C09156=1172.373,-59.206,-43.049,179.363,5.809,149.223
C09157=1172.378,-59.456,-43.037,179.360,5.808,149.223
C09158=1172.384,-59.705,-43.026,179.358,5.808,149.224
C09159=1172.389,-59.955,-43.015,179.356,5.808,149.225
C09160=1172.394,-60.205,-43.003,179.354,5.807,149.225
C09161=1172.400,-60.454,-42.993,179.351,5.807,149.226
C09162=1172.404,-60.704,-42.982,179.349,5.806,149.227
C09163=1172.410,-60.953,-42.971,179.347,5.807,149.227
C09164=1172.415,-61.203,-42.960,179.344,5.806,149.228
C09165=1172.420,-61.453,-42.948,179.342,5.805,149.228
C09166=1172.426,-61.702,-42.938,179.339,5.805,149.229
C09167=1172.430,-61.952,-42.927,179.337,5.805,149.230
C09168=1172.436,-62.203,-42.916,179.335,5.805,149.230
C09169=1172.441,-62.452,-42.905,179.333,5.804,149.231
C09170=1172.446,-62.702,-42.894,179.331,5.804,149.232
C09171=1172.452,-62.951,-42.883,179.328,5.803,149.232
C09172=1172.456,-63.200,-42.872,179.326,5.803,149.233
C09173=1172.462,-63.451,-42.861,179.323,5.803,149.233
C09174=1172.467,-63.700,-42.850,179.321,5.803,149.234
C09175=1172.472,-63.950,-42.839,179.319,5.802,149.235
C09176=1172.478,-64.199,-42.828,179.317,5.801,149.235
C09177=1172.483,-64.449,-42.818,179.314,5.801,149.236
C09178=1172.488,-64.699,-42.806,179.312,5.801,149.236
C09179=1172.494,-64.949,-42.796,179.310,5.801,149.237
C09180=1172.498,-65.198,-42.784,179.307,5.800,149.238
C09181=1172.504,-65.448,-42.774,179.305,5.800,149.238
C09182=1172.509,-65.698,-42.764,179.303,5.800,149.239
C09183=1172.515,-65.947,-42.752,179.301,5.799,149.239
C09184=1172.520,-66.198,-42.742,179.298,5.799,149.240
C09185=1172.525,-66.447,-42.730,179.296,5.799,149.241
C09186=1172.530,-66.697,-42.720,179.294,5.798,149.241
C09187=1172.535,-66.946,-42.709,179.291,5.798,149.242
C09188=1172.541,-67.196,-42.699,179.289,5.798,149.242
C09189=1172.546,-67.446,-42.688,179.287,5.797,149.243
C09190=1172.552,-67.695,-42.677,179.284,5.796,149.244
C09191=1172.557,-67.946,-42.666,179.282,5.797,149.244
C09192=1172.562,-68.195,-42.655,179.280,5.796,149.245
C09193=1172.567,-68.445,-42.644,179.278,5.796,149.245
C09194=1172.573,-68.694,-42.634,179.275,5.795,149.246
C09195=1172.577,-68.944,-42.623,179.273,5.795,149.247
C09196=1172.583,-69.194,-42.613,179.271,5.795,149.247
C09197=1172.588,-69.444,-42.602,179.268,5.794,149.248
C09198=1172.593,-69.693,-42.591,179.266,5.794,149.249
C09199=1172.598,-69.943,-42.581,179.264,5.794,149.249
C09200=1172.605,-70.193,-42.570,179.261,5.793,149.250
C09201=1172.609,-70.442,-42.559,179.259,5.794,149.250
C09202=1172.615,-70.692,-42.548,179.257,5.793,149.251
C09203=1172.620,-70.942,-42.538,179.255,5.792,149.252
C09204=1172.625,-71.191,-42.527,179.253,5.792,149.252
C09205=1172.630,-71.441,-42.516,179.250,5.792,149.253
C09206=1172.636,-71.691,-42.506,179.248,5.791,149.253
C09207=1172.641,-71.941,-42.495,179.246,5.792,149.254
C09208=1172.646,-72.190,-42.485,179.244,5.791,149.254
C09209=1172.651,-72.440,-42.474,179.241,5.790,149.255
C09210=1172.657,-72.690,-42.464,179.238,5.790,149.256
C09211=1172.661,-72.940,-42.452,179.237,5.790,149.256
C09212=1172.667,-73.189,-42.442,179.234,5.790,149.257
C09213=1172.672,-73.439,-42.432,179.232,5.789,149.258
C09214=1172.677,-73.689,-42.422,179.230,5.789,149.258
C09215=1172.683,-73.938,-42.411,179.228,5.788,149.259
C09216=1172.688,-74.188,-42.400,179.225,5.788,149.259
C09217=1172.693,-74.438,-42.390,179.224,5.788,149.260
C09218=1172.698,-74.688,-42.379,179.221,5.788,149.261
C09219=1172.704,-74.937,-42.369,179.219,5.787,149.261
C09220=1172.709,-75.188,-42.358,179.217,5.787,149.262
C09221=1172.714,-75.437,-42.348,179.214,5.787,149.263
C09222=1172.720,-75.708,-42.336,179.212,5.786,149.263
C09223=1172.726,-75.979,-42.325,179.209,5.786,149.264
C09224=1172.732,-76.250,-42.314,179.207,5.786,149.264
C09225=1172.737,-76.521,-42.302,179.204,5.786,149.265
C09226=1172.742,-76.771,-42.292,179.202,5.785,149.266
C09227=1172.748,-77.020,-42.282,179.200,5.785,149.266
C09228=1172.753,-77.270,-42.271,179.198,5.784,149.267
C09229=1172.759,-77.520,-42.261,179.195,5.784,149.268
C09230=1172.764,-77.770,-42.250,179.194,5.784,149.268
C09231=1172.769,-78.020,-42.240,179.191,5.784,149.269
C09232=1172.775,-78.269,-42.230,179.189,5.783,149.269
C09233=1172.779,-78.519,-42.219,179.187,5.783,149.270
C09234=1172.785,-78.768,-42.209,179.184,5.783,149.270
C09235=1172.790,-79.019,-42.198,179.182,5.782,149.271
C09236=1172.796,-79.268,-42.188,179.180,5.783,149.272
C09237=1172.801,-79.518,-42.178,179.177,5.782,149.272
C09238=1172.805,-79.768,-42.168,179.175,5.781,149.273
C09239=1172.811,-80.017,-42.157,179.173,5.781,149.274
C09240=1172.817,-80.267,-42.147,179.171,5.781,149.274
C09241=1172.822,-80.517,-42.137,179.168,5.780,149.275
C09242=1172.827,-80.767,-42.126,179.166,5.781,149.275
C09243=1172.833,-81.016,-42.116,179.164,5.780,149.276
C09244=1172.838,-81.266,-42.106,179.161,5.779,149.277
C09245=1172.843,-81.516,-42.096,179.160,5.779,149.277
C09246=1172.848,-81.766,-42.085,179.157,5.779,149.278
C09247=1172.853,-82.015,-42.075,179.155,5.778,149.278
C09248=1172.859,-82.265,-42.065,179.153,5.779,149.279
C09249=1172.864,-82.515,-42.054,179.151,5.778,149.279
C09250=1172.870,-82.765,-42.044,179.149,5.778,149.280
C09251=1172.874,-83.014,-42.035,179.146,5.777,149.281
C09252=1172.879,-83.264,-42.024,179.144,5.777,149.281
C09253=1172.885,-83.514,-42.014,179.142,5.777,149.282
C09254=1172.891,-83.763,-42.004,179.139,5.777,149.283
C09255=1172.896,-84.013,-41.993,179.137,5.776,149.283
C09256=1172.900,-84.263,-41.983,179.135,5.776,149.284
C09257=1172.906,-84.512,-41.973,179.133,5.776,149.284
C09258=1172.912,-84.762,-41.963,179.130,5.775,149.285
C09259=1172.917,-85.012,-41.952,179.128,5.775,149.286
C09260=1172.922,-85.262,-41.943,179.126,5.775,149.286
C09261=1172.927,-85.511,-41.933,179.124,5.775,149.287
C09262=1172.932,-85.762,-41.923,179.122,5.774,149.287
C09263=1172.938,-86.011,-41.913,179.119,5.774,149.288
C09264=1172.944,-86.261,-41.902,179.118,5.774,149.289
C09265=1172.948,-86.510,-41.893,179.115,5.774,149.289
C09266=1172.953,-86.760,-41.882,179.113,5.773,149.290
C09267=1172.959,-87.010,-41.872,179.111,5.773,149.290
C09268=1172.964,-87.260,-41.863,179.108,5.772,149.291
C09269=1172.969,-87.510,-41.852,179.106,5.773,149.292
C09270=1172.975,-87.759,-41.842,179.104,5.772,149.292
C09271=1172.980,-88.009,-41.832,179.101,5.772,149.293
C09272=1172.985,-88.258,-41.822,179.100,5.772,149.293
C09273=1172.990,-88.508,-41.812,179.097,5.771,149.294
C09274=1172.996,-88.759,-41.802,179.096,5.771,149.294
C09275=1173.001,-89.008,-41.793,179.093,5.771,149.295
C09276=1173.007,-89.257,-41.783,179.091,5.770,149.296
C09277=1173.012,-89.508,-41.772,179.089,5.770,149.296
C09278=1173.016,-89.757,-41.762,179.086,5.770,149.297
C09279=1173.022,-90.007,-41.753,179.084,5.769,149.298
C09280=1173.028,-90.257,-41.743,179.082,5.769,149.298
C09281=1173.032,-90.507,-41.733,179.080,5.769,149.299
C09282=1173.038,-90.756,-41.722,179.078,5.769,149.299
C09283=1173.044,-91.006,-41.713,179.075,5.769,149.300
C09284=1173.049,-91.255,-41.703,179.073,5.768,149.300
C09285=1173.054,-91.505,-41.693,179.071,5.768,149.301
C09286=1173.059,-91.755,-41.683,179.069,5.767,149.302
C09287=1173.064,-92.005,-41.674,179.067,5.768,149.302
C09288=1173.070,-92.255,-41.663,179.065,5.767,149.303
C09289=1173.076,-92.504,-41.653,179.062,5.767,149.304
C09290=1173.081,-92.754,-41.644,179.060,5.767,149.304
C09291=1173.086,-93.004,-41.634,179.058,5.766,149.305
C09292=1173.091,-93.253,-41.624,179.056,5.766,149.305
C09293=1173.097,-93.504,-41.615,179.053,5.766,149.306
C09294=1173.102,-93.753,-41.604,179.051,5.765,149.306
C09295=1173.107,-94.002,-41.595,179.049,5.765,149.307
C09296=1173.112,-94.253,-41.585,179.047,5.765,149.308
C09297=1173.118,-94.503,-41.575,179.045,5.765,149.308
C09298=1173.123,-94.752,-41.565,179.043,5.764,149.309
C09299=1173.129,-95.002,-41.556,179.040,5.764,149.310
C09300=1173.133,-95.251,-41.546,179.038,5.764,149.310
C09301=1173.139,-95.501,-41.536,179.036,5.764,149.311
C09302=1173.144,-95.752,-41.527,179.034,5.764,149.311
C09303=1173.149,-96.001,-41.516,179.032,5.763,149.312
C09304=1173.155,-96.251,-41.506,179.030,5.763,149.312
C09305=1173.160,-96.500,-41.497,179.028,5.762,149.313
C09306=1173.166,-96.750,-41.487,179.025,5.762,149.314
C09307=1173.171,-97.000,-41.478,179.023,5.762,149.314
C09308=1173.176,-97.249,-41.468,179.021,5.762,149.315
C09309=1173.182,-97.499,-41.459,179.019,5.762,149.315
C09310=1173.187,-97.750,-41.448,179.016,5.761,149.316
C09311=1173.191,-97.999,-41.439,179.014,5.760,149.316
C09312=1173.197,-98.249,-41.429,179.012,5.761,149.317
C09313=1173.202,-98.498,-41.420,179.010,5.760,149.318
C09314=1173.208,-98.748,-41.410,179.008,5.761,149.318
C09315=1173.213,-98.998,-41.401,179.006,5.760,149.319
C09316=1173.219,-99.248,-41.391,179.004,5.760,149.320
C09317=1173.224,-99.497,-41.382,179.001,5.759,149.320
C09318=1173.230,-99.747,-41.372,178.999,5.759,149.321
C09319=1173.234,-99.997,-41.362,178.997,5.759,149.321
C09320=1173.240,-100.247,-41.353,178.995,5.758,149.322
C09321=1173.245,-100.496,-41.343,178.993,5.759,149.322
C09322=1173.251,-100.747,-41.333,178.991,5.758,149.323
C09323=1173.255,-100.996,-41.324,178.989,5.758,149.324
C09324=1173.261,-101.246,-41.314,178.986,5.758,149.324
C09325=1173.266,-101.495,-41.305,178.984,5.757,149.325
C09326=1173.272,-101.767,-41.295,178.982,5.757,149.325
C09327=1173.278,-102.039,-41.284,178.979,5.757,149.326
C09328=1173.283,-102.311,-41.273,178.977,5.756,149.327
C09329=1173.289,-102.583,-41.264,178.975,5.756,149.327
C09330=1173.295,-102.832,-41.255,178.972,5.756,149.328
C09331=1173.300,-103.082,-41.244,178.970,5.755,149.328
C09332=1173.305,-103.332,-41.235,178.968,5.756,149.329
C09333=1173.310,-103.582,-41.225,178.966,5.755,149.330
C09334=1173.316,-103.832,-41.216,178.964,5.755,149.330
C09335=1173.321,-104.081,-41.206,178.962,5.755,149.331
C09336=1173.326,-104.331,-41.197,178.960,5.755,149.332
C09337=1173.332,-104.581,-41.188,178.957,5.754,149.332
C09338=1173.337,-104.831,-41.178,178.956,5.754,149.333
C09339=1173.342,-105.081,-41.169,178.953,5.754,149.333
C09340=1173.347,-105.330,-41.160,178.951,5.753,149.334
C09341=1173.353,-105.580,-41.150,178.949,5.753,149.334
C09342=1173.358,-105.830,-41.141,178.947,5.753,149.335
C09343=1173.364,-106.080,-41.132,178.945,5.753,149.336
C09344=1173.369,-106.329,-41.122,178.942,5.752,149.336
C09345=1173.374,-106.579,-41.113,178.941,5.752,149.337
C09346=1173.380,-106.829,-41.104,178.938,5.752,149.337
C09347=1173.385,-107.078,-41.094,178.937,5.752,149.338
C09348=1173.390,-107.328,-41.085,178.934,5.752,149.339
C09349=1173.396,-107.578,-41.076,178.932,5.751,149.339
C09350=1173.401,-107.828,-41.066,178.930,5.751,149.340
C09351=1173.406,-108.077,-41.057,178.927,5.750,149.340
C09352=1173.412,-108.328,-41.048,178.926,5.750,149.341
C09353=1173.417,-108.577,-41.038,178.923,5.750,149.341
C09354=1173.422,-108.827,-41.029,178.922,5.750,149.342
C09355=1173.428,-109.077,-41.019,178.919,5.750,149.343
C09356=1173.433,-109.327,-41.011,178.917,5.750,149.343
C09357=1173.438,-109.576,-41.001,178.915,5.749,149.344
C09358=1173.443,-109.826,-40.992,178.913,5.749,149.344
C09359=1173.449,-110.076,-40.983,178.911,5.749,149.345
C09360=1173.454,-110.326,-40.974,178.909,5.749,149.345
C09361=1173.459,-110.575,-40.964,178.906,5.748,149.346
C09362=1173.465,-110.825,-40.955,178.904,5.748,149.347
C09363=1173.470,-111.075,-40.946,178.902,5.748,149.347
C09364=1173.475,-111.325,-40.937,178.900,5.748,149.348
C09365=1173.480,-111.575,-40.928,178.898,5.748,149.348
C09366=1173.486,-111.824,-40.918,178.896,5.747,149.349
C09367=1173.491,-112.074,-40.909,178.894,5.747,149.350
C09368=1173.497,-112.323,-40.900,178.891,5.746,149.350
C09369=1173.502,-112.573,-40.891,178.889,5.747,149.351
C09370=1173.508,-112.823,-40.882,178.887,5.746,149.351
C09371=1173.513,-113.073,-40.873,178.886,5.746,149.352
C09372=1173.518,-113.322,-40.863,178.883,5.746,149.352
C09373=1173.523,-113.572,-40.854,178.881,5.746,149.353
C09374=1173.529,-113.822,-40.845,178.879,5.745,149.354
C09375=1173.534,-114.072,-40.836,178.877,5.745,149.354
C09376=1173.539,-114.322,-40.827,178.875,5.745,149.355
C09377=1173.545,-114.572,-40.818,178.873,5.745,149.355
C09378=1173.550,-114.822,-40.809,178.871,5.744,149.356
C09379=1173.555,-115.071,-40.799,178.868,5.745,149.357
C09380=1173.561,-115.321,-40.791,178.866,5.744,149.357
C09381=1173.566,-115.570,-40.782,178.864,5.743,149.358
C09382=1173.571,-115.820,-40.773,178.862,5.744,149.358
C09383=1173.577,-116.070,-40.764,178.860,5.743,149.359
C09384=1173.582,-116.320,-40.754,178.858,5.743,149.359
C09385=1173.588,-116.570,-40.746,178.856,5.742,149.360
C09386=1173.593,-116.820,-40.737,178.854,5.742,149.360
C09387=1173.598,-117.070,-40.728,178.851,5.742,149.361
C09388=1173.603,-117.320,-40.719,178.850,5.742,149.362
C09389=1173.609,-117.569,-40.710,178.847,5.741,149.362
C09390=1173.615,-117.819,-40.701,178.845,5.742,149.363
C09391=1173.620,-118.069,-40.692,178.843,5.741,149.363
C09392=1173.625,-118.319,-40.683,178.841,5.741,149.364
C09393=1173.630,-118.569,-40.674,178.839,5.741,149.365
C09394=1173.635,-118.818,-40.665,178.837,5.741,149.365
C09395=1173.641,-119.068,-40.656,178.835,5.740,149.366
C09396=1173.646,-119.317,-40.648,178.833,5.740,149.366
C09397=1173.652,-119.567,-40.639,178.831,5.740,149.367
C09398=1173.657,-119.817,-40.629,178.829,5.740,149.367
C09399=1173.663,-120.067,-40.621,178.827,5.739,149.368
C09400=1173.668,-120.317,-40.612,178.824,5.740,149.369
C09401=1173.673,-120.567,-40.603,178.822,5.739,149.369
C09402=1173.678,-120.817,-40.594,178.821,5.739,149.370
C09403=1173.684,-121.066,-40.585,178.818,5.739,149.370
C09404=1173.689,-121.316,-40.576,178.816,5.739,149.371
C09405=1173.694,-121.566,-40.567,178.814,5.738,149.371
C09406=1173.699,-121.816,-40.559,178.812,5.738,149.372
C09407=1173.705,-122.065,-40.550,178.810,5.737,149.372
C09408=1173.710,-122.314,-40.541,178.808,5.737,149.373
C09409=1173.716,-122.564,-40.532,178.806,5.737,149.374
C09410=1173.721,-122.814,-40.523,178.804,5.737,149.374
C09411=1173.726,-123.064,-40.514,178.801,5.737,149.375
C09412=1173.732,-123.314,-40.505,178.800,5.737,149.375
C09413=1173.737,-123.565,-40.497,178.798,5.736,149.376
C09414=1173.743,-123.814,-40.488,178.796,5.736,149.377
C09415=1173.748,-124.064,-40.479,178.793,5.736,149.377
C09416=1173.753,-124.314,-40.470,178.792,5.736,149.378
C09417=1173.759,-124.563,-40.462,178.789,5.735,149.378
C09418=1173.764,-124.813,-40.453,178.787,5.735,149.379
C09419=1173.769,-125.062,-40.444,178.785,5.735,149.379
C09420=1173.775,-125.312,-40.435,178.783,5.735,149.380
C09421=1173.780,-125.563,-40.427,178.781,5.734,149.380
C09422=1173.785,-125.813,-40.418,178.779,5.734,149.381
C09423=1173.791,-126.062,-40.410,178.777,5.734,149.382
C09424=1173.796,-126.312,-40.401,178.775,5.734,149.382
C09425=1173.801,-126.561,-40.392,178.773,5.733,149.383
C09426=1173.807,-126.811,-40.383,178.771,5.734,149.383
C09427=1173.813,-127.061,-40.375,178.769,5.734,149.384
C09428=1173.818,-127.311,-40.366,178.767,5.733,149.384
C09429=1173.823,-127.561,-40.357,178.765,5.733,149.385
C09430=1173.402,-127.572,-40.398,178.761,5.737,149.387
C09431=1173.397,-127.321,-40.407,178.763,5.736,149.386
C09432=1173.391,-127.072,-40.415,178.765,5.737,149.386
C09433=1173.386,-126.822,-40.424,178.767,5.737,149.385
C09434=1173.381,-126.573,-40.433,178.770,5.737,149.384
C09435=1173.375,-126.323,-40.442,178.771,5.737,149.384
C09436=1173.369,-126.073,-40.450,178.773,5.738,149.383
C09437=1173.364,-125.823,-40.459,178.775,5.737,149.383
C09438=1173.359,-125.573,-40.467,178.778,5.738,149.382
C09439=1173.354,-125.323,-40.476,178.779,5.738,149.382
C09440=1173.348,-125.074,-40.485,178.782,5.739,149.381
C09441=1173.343,-124.824,-40.494,178.784,5.739,149.381
C09442=1173.337,-124.574,-40.502,178.786,5.739,149.380
C09443=1173.332,-124.324,-40.511,178.788,5.739,149.379
C09444=1173.327,-124.074,-40.520,178.790,5.740,149.379
C09445=1173.321,-123.825,-40.528,178.792,5.740,149.378
C09446=1173.316,-123.575,-40.537,178.794,5.740,149.378
C09447=1173.310,-123.325,-40.547,178.796,5.740,149.377
C09448=1173.305,-123.075,-40.556,178.798,5.741,149.377
C09449=1173.300,-122.825,-40.565,178.800,5.740,149.376
C09450=1173.294,-122.576,-40.572,178.802,5.741,149.375
C09451=1173.289,-122.326,-40.581,178.804,5.741,149.375
C09452=1173.283,-122.076,-40.590,178.807,5.741,149.374
C09453=1173.278,-121.826,-40.599,178.808,5.741,149.374
C09454=1173.273,-121.576,-40.608,178.811,5.742,149.373
C09455=1173.267,-121.327,-40.616,178.813,5.742,149.373
C09456=1173.262,-121.077,-40.625,178.815,5.743,149.372
C09457=1173.257,-120.827,-40.634,178.817,5.742,149.371
C09458=1173.252,-120.578,-40.643,178.819,5.743,149.371
C09459=1173.247,-120.328,-40.652,178.821,5.743,149.370
C09460=1173.242,-120.078,-40.661,178.823,5.743,149.370
C09461=1173.236,-119.829,-40.669,178.825,5.743,149.369
C09462=1173.230,-119.579,-40.679,178.827,5.744,149.369
C09463=1173.225,-119.329,-40.688,178.829,5.744,149.368
C09464=1173.220,-119.079,-40.697,178.831,5.744,149.368
C09465=1173.214,-118.829,-40.706,178.833,5.744,149.367
C09466=1173.209,-118.579,-40.715,178.836,5.745,149.366
C09467=1173.204,-118.329,-40.723,178.837,5.745,149.366
C09468=1173.198,-118.080,-40.732,178.840,5.745,149.365
C09469=1173.193,-117.830,-40.741,178.842,5.745,149.365
C09470=1173.187,-117.580,-40.750,178.844,5.746,149.364
C09471=1173.182,-117.330,-40.759,178.846,5.745,149.363
C09472=1173.177,-117.080,-40.768,178.848,5.746,149.363
C09473=1173.172,-116.831,-40.777,178.850,5.746,149.362
C09474=1173.167,-116.581,-40.786,178.852,5.746,149.362
C09475=1173.161,-116.331,-40.795,178.854,5.746,149.361
C09476=1173.155,-116.081,-40.804,178.857,5.747,149.361
C09477=1173.150,-115.832,-40.813,178.858,5.747,149.360
C09478=1173.145,-115.582,-40.822,178.860,5.748,149.360
C09479=1173.140,-115.332,-40.831,178.862,5.747,149.359
C09480=1173.135,-115.083,-40.840,178.865,5.748,149.358
C09481=1173.129,-114.833,-40.849,178.867,5.747,149.358
C09482=1173.123,-114.583,-40.859,178.869,5.748,149.357
C09483=1173.118,-114.333,-40.868,178.870,5.748,149.357
C09484=1173.113,-114.083,-40.876,178.873,5.749,149.356
C09485=1173.108,-113.833,-40.885,178.875,5.749,149.356
C09486=1173.101,-113.584,-40.895,178.877,5.749,149.355
C09487=1173.097,-113.334,-40.904,178.879,5.749,149.354
C09488=1173.091,-113.084,-40.913,178.881,5.750,149.354
C09489=1173.086,-112.835,-40.922,178.883,5.749,149.353
C09490=1173.081,-112.585,-40.931,178.885,5.750,149.353
C09491=1173.075,-112.335,-40.940,178.888,5.750,149.352
C09492=1173.070,-112.085,-40.949,178.890,5.750,149.351
C09493=1173.065,-111.836,-40.959,178.892,5.751,149.351
C09494=1173.060,-111.586,-40.968,178.894,5.751,149.350
C09495=1173.054,-111.336,-40.977,178.896,5.752,149.350
C09496=1173.049,-111.086,-40.986,178.898,5.751,149.349
C09497=1173.044,-110.836,-40.995,178.901,5.752,149.349
C09498=1173.038,-110.586,-41.005,178.902,5.752,149.348
C09499=1173.033,-110.336,-41.014,178.905,5.752,149.347
C09500=1173.028,-110.087,-41.023,178.906,5.752,149.347
C09501=1173.023,-109.837,-41.032,178.909,5.753,149.346
C09502=1173.017,-109.587,-41.041,178.911,5.753,149.346
C09503=1173.012,-109.337,-41.051,178.913,5.753,149.345
C09504=1173.007,-109.087,-41.060,178.916,5.754,149.344
C09505=1173.001,-108.837,-41.069,178.917,5.754,149.344
C09506=1172.995,-108.588,-41.078,178.920,5.754,149.343
C09507=1172.990,-108.339,-41.088,178.921,5.754,149.343
C09508=1172.984,-108.089,-41.097,178.924,5.754,149.342
C09509=1172.979,-107.839,-41.106,178.926,5.754,149.342
C09510=1172.974,-107.590,-41.116,178.928,5.755,149.341
C09511=1172.968,-107.340,-41.125,178.930,5.755,149.340
C09512=1172.963,-107.090,-41.134,178.932,5.756,149.340
C09513=1172.958,-106.840,-41.144,178.934,5.755,149.339
C09514=1172.952,-106.590,-41.153,178.936,5.756,149.339
C09515=1172.947,-106.340,-41.162,178.939,5.756,149.338
C09516=1172.943,-106.090,-41.172,178.941,5.756,149.337
C09517=1172.937,-105.840,-41.181,178.943,5.757,149.337
C09518=1172.932,-105.590,-41.190,178.945,5.757,149.336
C09519=1172.927,-105.341,-41.200,178.947,5.757,149.336
C09520=1172.921,-105.091,-41.209,178.949,5.757,149.335
C09521=1172.916,-104.841,-41.218,178.951,5.758,149.335
C09522=1172.911,-104.592,-41.228,178.954,5.757,149.334
C09523=1172.905,-104.342,-41.237,178.956,5.758,149.333
C09524=1172.900,-104.092,-41.246,178.958,5.759,149.333
C09525=1172.894,-103.842,-41.257,178.960,5.758,149.332
C09526=1172.889,-103.593,-41.265,178.962,5.759,149.332
C09527=1172.884,-103.343,-41.275,178.964,5.759,149.331
C09528=1172.879,-103.093,-41.285,178.966,5.760,149.331
C09529=1172.873,-102.843,-41.293,178.969,5.759,149.330
C09530=1172.868,-102.594,-41.304,178.971,5.760,149.329
C09531=1172.862,-102.322,-41.314,178.973,5.760,149.329
C09532=1172.857,-102.050,-41.324,178.975,5.760,149.328
C09533=1172.851,-101.779,-41.334,178.978,5.761,149.327
C09534=1172.844,-101.507,-41.345,178.980,5.761,149.327
C09535=1172.840,-101.257,-41.354,178.982,5.761,149.326
C09536=1172.834,-101.007,-41.363,178.985,5.761,149.325
C09537=1172.829,-100.757,-41.374,178.986,5.761,149.325
C09538=1172.824,-100.507,-41.383,178.989,5.762,149.324
C09539=1172.819,-100.258,-41.393,178.991,5.763,149.324
C09540=1172.813,-100.008,-41.402,178.993,5.762,149.323
C09541=1172.808,-99.758,-41.412,178.995,5.763,149.323
C09542=1172.803,-99.509,-41.421,178.997,5.763,149.322
C09543=1172.797,-99.259,-41.431,179.000,5.763,149.321
C09544=1172.792,-99.009,-41.440,179.001,5.763,149.321
C09545=1172.786,-98.760,-41.450,179.004,5.764,149.320
C09546=1172.781,-98.510,-41.459,179.006,5.765,149.320
C09547=1172.776,-98.260,-41.470,179.008,5.764,149.319
C09548=1172.771,-98.010,-41.479,179.010,5.765,149.319
C09549=1172.765,-97.760,-41.489,179.012,5.764,149.318
C09550=1172.760,-97.510,-41.498,179.015,5.765,149.317
C09551=1172.755,-97.261,-41.508,179.017,5.765,149.317
C09552=1172.750,-97.011,-41.517,179.019,5.766,149.316
C09553=1172.744,-96.761,-41.527,179.022,5.766,149.315
C09554=1172.738,-96.512,-41.537,179.023,5.766,149.315
C09555=1172.734,-96.261,-41.547,179.026,5.766,149.314
C09556=1172.728,-96.012,-41.557,179.027,5.766,149.314
C09557=1172.723,-95.762,-41.566,179.030,5.767,149.313
C09558=1172.717,-95.512,-41.576,179.032,5.768,149.313
C09559=1172.713,-95.263,-41.586,179.034,5.768,149.312
C09560=1172.707,-95.013,-41.595,179.037,5.768,149.311
C09561=1172.701,-94.763,-41.605,179.038,5.768,149.311
C09562=1172.697,-94.513,-41.615,179.041,5.768,149.310
C09563=1172.691,-94.263,-41.625,179.043,5.769,149.310
C09564=1172.686,-94.014,-41.634,179.045,5.769,149.309
C09565=1172.680,-93.764,-41.644,179.047,5.769,149.308
C09566=1172.674,-93.514,-41.654,179.049,5.769,149.308
C09567=1172.670,-93.264,-41.664,179.052,5.770,149.307
C09568=1172.665,-93.015,-41.674,179.054,5.770,149.307
C09569=1172.659,-92.765,-41.683,179.056,5.770,149.306
C09570=1172.654,-92.515,-41.693,179.059,5.771,149.305
C09571=1172.648,-92.266,-41.703,179.060,5.771,149.305
C09572=1172.644,-92.015,-41.713,179.063,5.771,149.304
C09573=1172.638,-91.766,-41.723,179.065,5.772,149.304
C09574=1172.633,-91.517,-41.733,179.067,5.771,149.303
C09575=1172.628,-91.267,-41.743,179.069,5.772,149.303
C09576=1172.622,-91.017,-41.752,179.071,5.772,149.302
C09577=1172.617,-90.767,-41.762,179.074,5.772,149.301
C09578=1172.612,-90.517,-41.772,179.076,5.773,149.301
C09579=1172.606,-90.268,-41.783,179.078,5.773,149.300
C09580=1172.601,-90.018,-41.792,179.080,5.773,149.299
C09581=1172.596,-89.768,-41.802,179.082,5.773,149.299
C09582=1172.591,-89.518,-41.812,179.085,5.774,149.298
C09583=1172.586,-89.269,-41.822,179.087,5.774,149.298
C09584=1172.580,-89.019,-41.831,179.089,5.774,149.297
C09585=1172.574,-88.769,-41.842,179.091,5.775,149.297
C09586=1172.569,-88.519,-41.852,179.093,5.774,149.296
C09587=1172.564,-88.270,-41.862,179.095,5.775,149.295
C09588=1172.559,-88.020,-41.872,179.098,5.776,149.295
C09589=1172.553,-87.770,-41.882,179.100,5.776,149.294
C09590=1172.549,-87.520,-41.892,179.102,5.776,149.293
C09591=1172.543,-87.271,-41.902,179.105,5.777,149.293
C09592=1172.537,-87.021,-41.912,179.107,5.776,149.292
C09593=1172.532,-86.771,-41.923,179.109,5.777,149.292
C09594=1172.527,-86.522,-41.932,179.111,5.777,149.291
C09595=1172.522,-86.272,-41.942,179.113,5.777,149.291
C09596=1172.516,-86.022,-41.952,179.116,5.778,149.290
C09597=1172.512,-85.772,-41.962,179.117,5.778,149.289
C09598=1172.506,-85.522,-41.972,179.120,5.778,149.289
C09599=1172.501,-85.273,-41.982,179.122,5.779,149.288
C09600=1172.496,-85.023,-41.993,179.124,5.779,149.287
C09601=1172.490,-84.773,-42.003,179.127,5.779,149.287
C09602=1172.485,-84.524,-42.013,179.129,5.779,149.286
C09603=1172.479,-84.274,-42.023,179.131,5.780,149.286
C09604=1172.474,-84.024,-42.033,179.134,5.780,149.285
C09605=1172.469,-83.775,-42.044,179.135,5.780,149.285
C09606=1172.464,-83.525,-42.053,179.138,5.781,149.284
C09607=1172.459,-83.275,-42.064,179.140,5.781,149.283
C09608=1172.453,-83.025,-42.073,179.142,5.781,149.283
C09609=1172.448,-82.775,-42.084,179.144,5.782,149.282
C09610=1172.443,-82.525,-42.094,179.147,5.782,149.282
C09611=1172.438,-82.276,-42.104,179.148,5.782,149.281
C09612=1172.432,-82.026,-42.114,179.151,5.783,149.280
C09613=1172.427,-81.776,-42.124,179.153,5.783,149.280
C09614=1172.421,-81.527,-42.135,179.155,5.783,149.279
C09615=1172.416,-81.277,-42.145,179.158,5.784,149.279
C09616=1172.411,-81.027,-42.155,179.160,5.783,149.278
C09617=1172.405,-80.777,-42.166,179.162,5.784,149.277
C09618=1172.400,-80.528,-42.175,179.165,5.785,149.277
C09619=1172.395,-80.278,-42.186,179.167,5.784,149.276
C09620=1172.390,-80.028,-42.196,179.169,5.785,149.276
C09621=1172.385,-79.779,-42.207,179.172,5.785,149.275
C09622=1172.380,-79.529,-42.218,179.173,5.785,149.274
C09623=1172.374,-79.279,-42.228,179.176,5.786,149.274
C09624=1172.369,-79.029,-42.238,179.178,5.786,149.273
C09625=1172.363,-78.780,-42.249,179.180,5.786,149.272
C09626=1172.358,-78.530,-42.258,179.182,5.787,149.272
C09627=1172.353,-78.280,-42.269,179.185,5.787,149.271
C09628=1172.348,-78.031,-42.279,179.186,5.787,149.271
C09629=1172.343,-77.780,-42.290,179.189,5.788,149.270
C09630=1172.337,-77.531,-42.300,179.191,5.788,149.270
C09631=1172.332,-77.281,-42.310,179.193,5.788,149.269
C09632=1172.327,-77.031,-42.321,179.196,5.788,149.268
C09633=1172.321,-76.782,-42.331,179.198,5.789,149.268
C09634=1172.316,-76.532,-42.342,179.200,5.789,149.267
C09635=1172.311,-76.261,-42.353,179.203,5.790,149.267
C09636=1172.305,-75.990,-42.364,179.205,5.790,149.266
C09637=1172.299,-75.718,-42.376,179.208,5.790,149.265
C09638=1172.293,-75.448,-42.387,179.210,5.790,149.264
C09639=1172.288,-75.198,-42.398,179.212,5.791,149.264
C09640=1172.283,-74.948,-42.408,179.215,5.791,149.263
C09641=1172.277,-74.699,-42.418,179.216,5.791,149.263
C09642=1172.272,-74.449,-42.429,179.219,5.792,149.262
C09643=1172.267,-74.200,-42.439,179.221,5.792,149.262
C09644=1172.262,-73.949,-42.450,179.223,5.792,149.261
C09645=1172.256,-73.700,-42.460,179.226,5.793,149.260
C09646=1172.251,-73.450,-42.471,179.228,5.793,149.260
C09647=1172.246,-73.200,-42.481,179.231,5.794,149.259
C09648=1172.241,-72.950,-42.492,179.233,5.794,149.258
C09649=1172.235,-72.701,-42.503,179.235,5.794,149.258
C09650=1172.230,-72.451,-42.513,179.237,5.795,149.257
C09651=1172.225,-72.201,-42.523,179.239,5.794,149.257
C09652=1172.219,-71.952,-42.534,179.242,5.795,149.256
C09653=1172.214,-71.702,-42.545,179.244,5.796,149.255
C09654=1172.209,-71.452,-42.555,179.246,5.796,149.255
C09655=1172.204,-71.203,-42.566,179.249,5.796,149.254
C09656=1172.198,-70.953,-42.577,179.251,5.797,149.254
C09657=1172.193,-70.703,-42.588,179.253,5.796,149.253
C09658=1172.187,-70.453,-42.598,179.256,5.797,149.252
C09659=1172.183,-70.203,-42.609,179.258,5.798,149.252
C09660=1172.177,-69.954,-42.619,179.260,5.797,149.251
C09661=1172.172,-69.704,-42.630,179.262,5.798,149.251
C09662=1172.167,-69.455,-42.641,179.265,5.798,149.250
C09663=1172.162,-69.205,-42.651,179.267,5.799,149.249
C09664=1172.156,-68.955,-42.662,179.269,5.799,149.249
C09665=1172.151,-68.705,-42.673,179.271,5.800,149.248
C09666=1172.146,-68.456,-42.683,179.274,5.800,149.248
C09667=1172.141,-68.206,-42.694,179.276,5.800,149.247
C09668=1172.135,-67.956,-42.705,179.278,5.800,149.246
C09669=1172.130,-67.706,-42.716,179.281,5.801,149.246
C09670=1172.124,-67.457,-42.727,179.282,5.801,149.245
C09671=1172.119,-67.207,-42.737,179.285,5.801,149.244
C09672=1172.114,-66.958,-42.748,179.287,5.802,149.244
C09673=1172.109,-66.708,-42.759,179.290,5.802,149.243
C09674=1172.104,-66.458,-42.769,179.292,5.802,149.243
C09675=1172.098,-66.208,-42.781,179.294,5.803,149.242
C09676=1172.093,-65.958,-42.792,179.297,5.803,149.241
C09677=1172.088,-65.709,-42.802,179.298,5.803,149.241
C09678=1172.083,-65.459,-42.813,179.301,5.804,149.240
C09679=1172.078,-65.210,-42.824,179.303,5.804,149.240
C09680=1172.073,-64.960,-42.835,179.305,5.804,149.239
C09681=1172.067,-64.710,-42.846,179.308,5.804,149.238
C09682=1172.061,-64.460,-42.857,179.310,5.805,149.238
C09683=1172.056,-64.210,-42.867,179.313,5.806,149.237
C09684=1172.051,-63.961,-42.878,179.314,5.806,149.237
C09685=1172.046,-63.711,-42.889,179.317,5.806,149.236
C09686=1172.040,-63.462,-42.900,179.319,5.807,149.235
C09687=1172.035,-63.212,-42.911,179.322,5.807,149.235
C09688=1172.030,-62.962,-42.922,179.324,5.807,149.234
C09689=1172.025,-62.713,-42.933,179.326,5.808,149.234
C09690=1172.020,-62.463,-42.944,179.329,5.808,149.233
C09691=1172.014,-62.213,-42.955,179.330,5.808,149.232
C09692=1172.009,-61.963,-42.966,179.333,5.809,149.232
C09693=1172.004,-61.713,-42.977,179.335,5.809,149.231
C09694=1171.999,-61.464,-42.987,179.338,5.810,149.230
C09695=1171.993,-61.214,-42.999,179.340,5.809,149.230
C09696=1171.988,-60.964,-43.010,179.342,5.810,149.229
C09697=1171.983,-60.715,-43.021,179.345,5.811,149.229
C09698=1171.978,-60.465,-43.032,179.347,5.811,149.228
C09699=1171.972,-60.215,-43.043,179.349,5.811,149.227
C09700=1171.967,-59.966,-43.054,179.351,5.812,149.227
C09701=1171.963,-59.716,-43.065,179.354,5.812,149.226
C09702=1171.957,-59.467,-43.075,179.356,5.812,149.226
C09703=1171.952,-59.217,-43.087,179.358,5.813,149.225
C09704=1171.947,-58.966,-43.098,179.361,5.813,149.224
C09705=1171.941,-58.717,-43.109,179.363,5.814,149.224
C09706=1171.936,-58.467,-43.121,179.365,5.813,149.223
C09707=1171.931,-58.217,-43.131,179.368,5.814,149.222
C09708=1171.926,-57.968,-43.142,179.370,5.815,149.222
C09709=1171.920,-57.718,-43.154,179.373,5.815,149.221
C09710=1171.915,-57.468,-43.165,179.374,5.815,149.221
C09711=1171.910,-57.219,-43.176,179.377,5.815,149.220
C09712=1171.905,-56.969,-43.187,179.379,5.816,149.220
C09713=1171.900,-56.720,-43.199,179.382,5.817,149.219
C09714=1171.894,-56.470,-43.209,179.384,5.816,149.218
C09715=1171.889,-56.220,-43.221,179.386,5.817,149.218
C09716=1171.884,-55.971,-43.232,179.389,5.818,149.217
C09717=1171.879,-55.720,-43.243,179.391,5.818,149.217
C09718=1171.873,-55.471,-43.254,179.393,5.818,149.216
C09719=1171.868,-55.221,-43.266,179.396,5.818,149.215
C09720=1171.864,-54.972,-43.277,179.398,5.819,149.215
C09721=1171.857,-54.722,-43.288,179.401,5.820,149.214
C09722=1171.853,-54.472,-43.299,179.402,5.820,149.214
C09723=1171.847,-54.222,-43.311,179.405,5.820,149.213
C09724=1171.843,-53.973,-43.322,179.407,5.820,149.212
C09725=1171.837,-53.724,-43.333,179.410,5.821,149.212
C09726=1171.832,-53.473,-43.344,179.412,5.822,149.211
C09727=1171.827,-53.224,-43.355,179.414,5.822,149.210
C09728=1171.821,-52.974,-43.367,179.417,5.822,149.210
C09729=1171.816,-52.725,-43.378,179.419,5.822,149.209
C09730=1171.811,-52.475,-43.390,179.421,5.823,149.209
C09731=1171.806,-52.225,-43.401,179.424,5.823,149.208
C09732=1171.801,-51.975,-43.412,179.426,5.824,149.207
C09733=1171.795,-51.726,-43.424,179.428,5.824,149.207
C09734=1171.790,-51.476,-43.435,179.431,5.825,149.206
C09735=1171.785,-51.226,-43.447,179.433,5.825,149.205
C09736=1171.780,-50.977,-43.458,179.435,5.825,149.205
C09737=1171.774,-50.727,-43.470,179.437,5.826,149.204
C09738=1171.769,-50.478,-43.481,179.440,5.826,149.204
C09739=1171.764,-50.207,-43.493,179.443,5.827,149.203
C09740=1171.758,-49.936,-43.505,179.445,5.827,149.202
C09741=1171.752,-49.666,-43.518,179.448,5.828,149.202
C09742=1171.747,-49.395,-43.530,179.450,5.827,149.201
C09743=1171.741,-49.146,-43.541,179.452,5.828,149.200
C09744=1171.736,-48.896,-43.553,179.455,5.829,149.200
C09745=1171.731,-48.647,-43.564,179.457,5.829,149.199
C09746=1171.726,-48.397,-43.576,179.460,5.830,149.198
C09747=1171.720,-48.147,-43.588,179.462,5.830,149.198
C09748=1171.716,-47.897,-43.599,179.464,5.830,149.197
C09749=1171.710,-47.648,-43.611,179.466,5.831,149.197
C09750=1171.705,-47.398,-43.622,179.469,5.831,149.196
C09751=1171.700,-47.148,-43.634,179.472,5.832,149.195
C09752=1171.695,-46.899,-43.645,179.473,5.832,149.195
C09753=1171.689,-46.649,-43.657,179.476,5.832,149.194
C09754=1171.684,-46.400,-43.668,179.478,5.833,149.194
C09755=1171.679,-46.150,-43.680,179.481,5.833,149.193
C09756=1171.673,-45.900,-43.692,179.483,5.834,149.192
C09757=1171.669,-45.650,-43.703,179.485,5.834,149.192
C09758=1171.663,-45.400,-43.715,179.488,5.834,149.191
C09759=1171.659,-45.151,-43.726,179.490,5.835,149.191
C09760=1171.652,-44.902,-43.738,179.493,5.835,149.190
C09761=1171.647,-44.652,-43.750,179.495,5.836,149.189
C09762=1171.642,-44.402,-43.761,179.497,5.836,149.189
C09763=1171.637,-44.152,-43.773,179.499,5.836,149.188
C09764=1171.633,-43.903,-43.785,179.502,5.837,149.188
C09765=1171.627,-43.653,-43.797,179.504,5.837,149.187
C09766=1171.622,-43.403,-43.809,179.507,5.838,149.186
C09767=1171.617,-43.154,-43.820,179.509,5.838,149.186
C09768=1171.611,-42.904,-43.832,179.511,5.838,149.185
C09769=1171.606,-42.654,-43.843,179.514,5.839,149.184
C09770=1171.601,-42.405,-43.855,179.516,5.840,149.184
C09771=1171.595,-42.155,-43.867,179.519,5.840,149.183
C09772=1171.590,-41.905,-43.879,179.521,5.841,149.183
C09773=1171.586,-41.656,-43.890,179.523,5.840,149.182
C09774=1171.580,-41.406,-43.902,179.526,5.841,149.181
C09775=1171.575,-41.156,-43.914,179.528,5.842,149.181
C09776=1171.570,-40.906,-43.926,179.531,5.842,149.180
C09777=1171.565,-40.656,-43.937,179.533,5.843,149.180
C09778=1171.559,-40.407,-43.950,179.535,5.842,149.179
C09779=1171.554,-40.158,-43.961,179.537,5.843,149.178
C09780=1171.549,-39.908,-43.973,179.540,5.844,149.178
C09781=1171.543,-39.658,-43.985,179.542,5.844,149.177
C09782=1171.539,-39.409,-43.996,179.544,5.845,149.177
C09783=1171.534,-39.159,-44.009,179.547,5.845,149.176
C09784=1171.528,-38.909,-44.020,179.549,5.845,149.175
C09785=1171.523,-38.659,-44.032,179.551,5.846,149.175
C09786=1171.518,-38.410,-44.044,179.554,5.846,149.174
C09787=1171.513,-38.161,-44.056,179.557,5.847,149.173
C09788=1171.507,-37.911,-44.068,179.559,5.848,149.173
C09789=1171.502,-37.661,-44.080,179.562,5.848,149.172
C09790=1171.498,-37.412,-44.092,179.563,5.848,149.172
C09791=1171.492,-37.162,-44.104,179.566,5.848,149.171
C09792=1171.487,-36.912,-44.116,179.568,5.849,149.170
C09793=1171.481,-36.662,-44.128,179.571,5.850,149.170
C09794=1171.476,-36.413,-44.140,179.573,5.850,149.169
C09795=1171.471,-36.163,-44.152,179.576,5.851,149.169
C09796=1171.466,-35.913,-44.163,179.578,5.851,149.168
C09797=1171.461,-35.664,-44.176,179.580,5.851,149.167
C09798=1171.456,-35.414,-44.188,179.582,5.852,149.167
C09799=1171.450,-35.164,-44.200,179.585,5.852,149.166
C09800=1171.446,-34.915,-44.212,179.588,5.853,149.165
C09801=1171.440,-34.665,-44.224,179.590,5.853,149.165
C09802=1171.435,-34.416,-44.236,179.593,5.854,149.164
C09803=1171.430,-34.166,-44.248,179.595,5.855,149.164
C09804=1171.424,-33.916,-44.260,179.597,5.854,149.163
C09805=1171.419,-33.666,-44.273,179.600,5.855,149.162
C09806=1171.414,-33.416,-44.285,179.602,5.856,149.162
C09807=1171.409,-33.167,-44.297,179.604,5.856,149.161
C09808=1171.404,-32.917,-44.308,179.607,5.856,149.160
C09809=1171.398,-32.668,-44.320,179.609,5.857,149.160
C09810=1171.393,-32.418,-44.333,179.612,5.858,149.159
C09811=1171.388,-32.168,-44.345,179.613,5.858,149.159
C09812=1171.383,-31.919,-44.357,179.616,5.858,149.158
C09813=1171.377,-31.669,-44.369,179.619,5.859,149.157
C09814=1171.372,-31.420,-44.382,179.621,5.859,149.157
C09815=1171.368,-31.170,-44.393,179.624,5.860,149.156
C09816=1171.362,-30.921,-44.406,179.626,5.861,149.156
C09817=1171.357,-30.671,-44.418,179.628,5.861,149.155
C09818=1171.352,-30.422,-44.430,179.631,5.861,149.154
C09819=1171.346,-30.172,-44.442,179.633,5.861,149.154
C09820=1171.341,-29.922,-44.455,179.635,5.862,149.153
C09821=1171.336,-29.672,-44.467,179.638,5.862,149.152
C09822=1171.331,-29.422,-44.480,179.640,5.863,149.152
C09823=1171.326,-29.172,-44.492,179.643,5.864,149.151
C09824=1171.321,-28.923,-44.504,179.645,5.864,149.151
C09825=1171.315,-28.673,-44.516,179.648,5.865,149.150
C09826=1171.310,-28.424,-44.529,179.650,5.865,149.149
C09827=1171.305,-28.174,-44.541,179.652,5.865,149.149
C09828=1171.300,-27.925,-44.553,179.655,5.866,149.148
C09829=1171.295,-27.675,-44.566,179.657,5.866,149.148
C09830=1171.289,-27.425,-44.578,179.659,5.867,149.147
C09831=1171.284,-27.176,-44.590,179.662,5.867,149.146
C09832=1171.279,-26.925,-44.602,179.664,5.868,149.146
C09833=1171.274,-26.676,-44.615,179.667,5.869,149.145
C09834=1171.269,-26.427,-44.628,179.670,5.869,149.145
C09835=1171.264,-26.177,-44.640,179.672,5.870,149.144
C09836=1171.258,-25.927,-44.652,179.674,5.870,149.143
C09837=1171.253,-25.678,-44.665,179.677,5.870,149.143
C09838=1171.248,-25.428,-44.677,179.679,5.871,149.142
C09839=1171.243,-25.178,-44.690,179.681,5.871,149.142
C09840=1171.238,-24.929,-44.702,179.684,5.872,149.141
C09841=1171.233,-24.679,-44.714,179.686,5.873,149.140
C09842=1171.228,-24.430,-44.727,179.689,5.873,149.140
C09843=1171.223,-24.160,-44.740,179.692,5.873,149.139
C09844=1171.217,-23.890,-44.753,179.694,5.874,149.139
C09845=1171.211,-23.620,-44.767,179.696,5.875,149.138
C09846=1171.206,-23.350,-44.781,179.699,5.875,149.137
C09847=1171.201,-23.100,-44.793,179.702,5.876,149.136
C09848=1171.195,-22.851,-44.805,179.704,5.876,149.136
C09849=1171.190,-22.602,-44.818,179.707,5.877,149.135
C09850=1171.185,-22.353,-44.831,179.709,5.877,149.135
C09851=1171.180,-22.102,-44.843,179.711,5.878,149.134
C09852=1171.175,-21.852,-44.856,179.714,5.879,149.133
C09853=1171.169,-21.603,-44.869,179.716,5.879,149.133
C09854=1171.164,-21.354,-44.881,179.718,5.879,149.132
C09855=1171.159,-21.104,-44.893,179.721,5.879,149.132
C09856=1171.154,-20.854,-44.906,179.723,5.880,149.131
C09857=1171.149,-20.604,-44.919,179.726,5.881,149.130
C09858=1171.143,-20.355,-44.932,179.728,5.881,149.130
C09859=1171.138,-20.105,-44.944,179.731,5.882,149.129
C09860=1171.133,-19.856,-44.957,179.733,5.882,149.129
C09861=1171.128,-19.605,-44.969,179.735,5.883,149.128
C09862=1171.123,-19.356,-44.982,179.738,5.884,149.127
C09863=1171.118,-19.107,-44.995,179.741,5.884,149.127
C09864=1171.112,-18.857,-45.008,179.743,5.885,149.126
C09865=1171.108,-18.607,-45.021,179.746,5.885,149.125
C09866=1171.102,-18.358,-45.033,179.748,5.886,149.125
C09867=1171.097,-18.109,-45.046,179.750,5.887,149.124
C09868=1171.092,-17.859,-45.059,179.753,5.887,149.124
C09869=1171.087,-17.609,-45.071,179.755,5.887,149.123
C09870=1171.082,-17.359,-45.084,179.757,5.888,149.122
C09871=1171.076,-17.110,-45.097,179.760,5.888,149.122
C09872=1171.071,-16.860,-45.109,179.762,5.889,149.121
C09873=1171.067,-16.610,-45.122,179.765,5.889,149.121
C09874=1171.061,-16.361,-45.135,179.768,5.890,149.120
C09875=1171.056,-16.111,-45.148,179.770,5.891,149.119
C09876=1171.051,-15.862,-45.161,179.772,5.891,149.119
C09877=1171.046,-15.612,-45.173,179.775,5.892,149.118
C09878=1171.040,-15.362,-45.187,179.777,5.892,149.118
C09879=1171.035,-15.113,-45.199,179.780,5.893,149.117
C09880=1171.031,-14.863,-45.212,179.782,5.894,149.116
C09881=1171.026,-14.614,-45.225,179.785,5.894,149.116
C09882=1171.020,-14.364,-45.238,179.787,5.894,149.115
C09883=1171.015,-14.114,-45.251,179.790,5.895,149.115
C09884=1171.010,-13.865,-45.264,179.792,5.896,149.114
C09885=1171.004,-13.615,-45.277,179.794,5.897,149.113
C09886=1171.000,-13.365,-45.290,179.797,5.897,149.113
C09887=1170.995,-13.116,-45.302,179.800,5.897,149.112
C09888=1170.989,-12.867,-45.315,179.802,5.898,149.112
C09889=1170.984,-12.616,-45.329,179.804,5.899,149.111
C09890=1170.979,-12.367,-45.341,179.807,5.899,149.110
C09891=1170.974,-12.118,-45.354,179.809,5.899,149.110
C09892=1170.969,-11.867,-45.367,179.811,5.900,149.109
C09893=1170.964,-11.619,-45.381,179.814,5.900,149.109
C09894=1170.959,-11.369,-45.393,179.816,5.901,149.108
C09895=1170.953,-11.119,-45.407,179.819,5.901,149.107
C09896=1170.948,-10.870,-45.419,179.821,5.902,149.107
C09897=1170.942,-10.620,-45.433,179.824,5.903,149.106
C09898=1170.938,-10.370,-45.446,179.826,5.903,149.105
C09899=1170.933,-10.121,-45.458,179.829,5.904,149.105
C09900=1170.928,-9.871,-45.472,179.831,5.904,149.104
C09901=1170.923,-9.622,-45.485,179.833,5.905,149.104
C09902=1170.918,-9.372,-45.498,179.836,5.906,149.103
C09903=1170.912,-9.122,-45.511,179.839,5.906,149.102
C09904=1170.907,-8.873,-45.524,179.841,5.907,149.102
C09905=1170.902,-8.622,-45.537,179.844,5.907,149.101
C09906=1170.897,-8.374,-45.551,179.846,5.908,149.100
C09907=1170.892,-8.124,-45.563,179.848,5.909,149.100
C09908=1170.887,-7.874,-45.577,179.851,5.909,149.099
C09909=1170.882,-7.625,-45.589,179.853,5.910,149.099
C09910=1170.877,-7.375,-45.604,179.856,5.910,149.098
C09911=1170.872,-7.126,-45.616,179.858,5.911,149.097
C09912=1170.866,-6.876,-45.630,179.861,5.912,149.097
C09913=1170.861,-6.626,-45.642,179.863,5.912,149.096
C09914=1170.856,-6.377,-45.656,179.866,5.913,149.096
C09915=1170.851,-6.127,-45.669,179.868,5.913,149.095
C09916=1170.846,-5.878,-45.682,179.871,5.914,149.094
C09917=1170.841,-5.627,-45.696,179.873,5.915,149.094
C09918=1170.836,-5.379,-45.709,179.876,5.915,149.093
C09919=1170.831,-5.128,-45.722,179.878,5.916,149.093
C09920=1170.825,-4.879,-45.735,179.880,5.916,149.092
C09921=1170.820,-4.630,-45.749,179.883,5.917,149.091
C09922=1170.815,-4.380,-45.762,179.886,5.917,149.091
C09923=1170.810,-4.130,-45.775,179.888,5.918,149.090
C09924=1170.805,-3.881,-45.789,179.891,5.919,149.090
C09925=1170.799,-3.631,-45.802,179.893,5.919,149.089
C09926=1170.794,-3.381,-45.816,179.895,5.920,149.088
C09927=1170.789,-3.132,-45.829,179.898,5.920,149.088
C09928=1170.784,-2.882,-45.842,179.900,5.921,149.087
C09929=1170.779,-2.633,-45.856,179.903,5.922,149.087
C09930=1170.774,-2.383,-45.869,179.906,5.922,149.086
C09931=1170.769,-2.134,-45.882,179.908,5.923,149.085
C09932=1170.764,-1.884,-45.896,179.910,5.923,149.085
C09933=1170.759,-1.634,-45.909,179.913,5.924,149.084
C09934=1170.754,-1.385,-45.923,179.915,5.925,149.084
C09935=1170.748,-1.135,-45.936,179.918,5.925,149.083
C09936=1170.744,-0.886,-45.950,179.921,5.927,149.082
C09937=1170.738,-0.636,-45.963,179.923,5.927,149.082
C09938=1170.734,-0.387,-45.977,179.926,5.928,149.081
C09939=1170.728,-0.137,-45.990,179.928,5.929,149.081
C09940=1170.723,0.113,-46.004,179.931,5.929,149.080
C09941=1170.718,0.362,-46.017,179.933,5.930,149.079
C09942=1170.713,0.612,-46.031,179.936,5.930,149.079
C09943=1170.707,0.861,-46.044,179.938,5.931,149.078
C09944=1170.703,1.111,-46.058,179.940,5.932,149.078
C09945=1170.697,1.361,-46.072,179.943,5.932,149.077
C09946=1170.693,1.610,-46.085,179.946,5.933,149.076
C09947=1170.687,1.880,-46.099,179.948,5.933,149.076
C09948=1170.682,2.149,-46.114,179.951,5.934,149.075
C09949=1170.675,2.418,-46.129,179.954,5.935,149.074
C09950=1170.670,2.687,-46.144,179.956,5.936,149.074
C09951=1170.666,2.937,-46.157,179.959,5.936,149.073
C09952=1170.660,3.186,-46.171,179.961,5.937,149.073
C09953=1170.655,3.436,-46.185,179.964,5.937,149.072
C09954=1170.649,3.686,-46.198,179.966,5.938,149.071
C09955=1170.645,3.935,-46.212,179.969,5.939,149.071
C09956=1170.640,4.185,-46.226,179.971,5.939,149.070
C09957=1170.634,4.434,-46.239,179.974,5.940,149.070
C09958=1170.630,4.684,-46.253,179.976,5.940,149.069
C09959=1170.625,4.934,-46.267,179.978,5.941,149.068
C09960=1170.619,5.183,-46.280,179.981,5.942,149.068
C09961=1170.614,5.433,-46.295,179.984,5.942,149.067
C09962=1170.609,5.682,-46.307,179.986,5.943,149.067
C09963=1170.604,5.932,-46.322,179.989,5.944,149.066
C09964=1170.599,6.182,-46.336,179.991,5.945,149.065
C09965=1170.594,6.431,-46.350,179.994,5.946,149.065
C09966=1170.589,6.681,-46.363,179.997,5.946,149.064
C09967=1170.584,6.930,-46.377,179.999,5.947,149.064
C09968=1170.578,7.179,-46.391,-179.999,5.947,149.063
C09969=1170.573,7.430,-46.404,-179.996,5.948,149.062
C09970=1170.568,7.679,-46.418,-179.994,5.949,149.062
C09971=1170.563,7.928,-46.432,-179.991,5.949,149.061
C09972=1170.559,8.178,-46.446,-179.989,5.950,149.061
C09973=1170.553,8.427,-46.460,-179.986,5.950,149.060
C09974=1170.548,8.677,-46.474,-179.984,5.951,149.059
C09975=1170.543,8.927,-46.488,-179.981,5.952,149.059
C09976=1170.538,9.176,-46.501,-179.978,5.953,149.058
C09977=1170.533,9.425,-46.516,-179.976,5.954,149.058
C09978=1170.528,9.676,-46.529,-179.973,5.954,149.057
C09979=1170.523,9.925,-46.544,-179.971,5.955,149.056
C09980=1170.517,10.174,-46.557,-179.969,5.956,149.056
C09981=1170.512,10.424,-46.572,-179.966,5.956,149.055
C09982=1170.507,10.674,-46.586,-179.964,5.957,149.055
C09983=1170.502,10.922,-46.599,-179.961,5.957,149.054
C09984=1170.497,11.173,-46.613,-179.958,5.958,149.053
C09985=1170.492,11.422,-46.627,-179.956,5.959,149.053
C09986=1170.487,11.671,-46.641,-179.954,5.959,149.052
C09987=1170.482,11.921,-46.655,-179.950,5.960,149.052
C09988=1170.477,12.171,-46.670,-179.948,5.961,149.051
C09989=1170.472,12.421,-46.684,-179.946,5.962,149.050
C09990=1170.466,12.670,-46.698,-179.943,5.963,149.050
C09991=1170.461,12.919,-46.712,-179.941,5.963,149.049
C09992=1170.456,13.169,-46.726,-179.938,5.963,149.049
C09993=1170.452,13.418,-46.740,-179.936,5.964,149.048
C09994=1170.446,13.668,-46.753,-179.933,5.965,149.047
C09995=1170.441,13.918,-46.768,-179.931,5.966,149.047
C09996=1170.436,14.167,-46.782,-179.928,5.967,149.046
//INST
///DATE 2021/06/15 17:25
///ATTR SC,RW,RJ
////FRAME ROBOT
///GROUP1 RB1
NOP
MOVL C00000 V=800.0 PL=0
MOVL C00001 V=800.0 PL=0
MOVL C00002 V=800.0 PL=0
MOVL C00003 V=800.0 PL=0
MOVL C00004 V=800.0 PL=0
MOVL C00005 V=800.0 PL=0
MOVL C00006 V=800.0 PL=0
MOVL C00007 V=800.0 PL=0
MOVL C00008 V=800.0 PL=0
MOVL C00009 V=800.0 PL=0
MOVL C00010 V=800.0 PL=0
MOVL C00011 V=800.0 PL=0
MOVL C00012 V=800.0 PL=0
MOVL C00013 V=800.0 PL=0
MOVL C00014 V=800.0 PL=0
MOVL C00015 V=800.0 PL=0
MOVL C00016 V=800.0 PL=0
MOVL C00017 V=800.0 PL=0
MOVL C00018 V=800.0 PL=0
MOVL C00019 V=800.0 PL=0
MOVL C00020 V=800.0 PL=0
MOVL C00021 V=800.0 PL=0
MOVL C00022 V=800.0 PL=0
MOVL C00023 V=800.0 PL=0
MOVL C00024 V=800.0 PL=0
MOVL C00025 V=800.0 PL=0
MOVL C00026 V=800.0 PL=0
MOVL C00027 V=800.0 PL=0
MOVL C00028 V=800.0 PL=0
MOVL C00029 V=800.0 PL=0
MOVL C00030 V=800.0 PL=0
MOVL C00031 V=800.0 PL=0
MOVL C00032 V=800.0 PL=0
MOVL C00033 V=800.0 PL=0
MOVL C00034 V=800.0 PL=0
MOVL C00035 V=800.0 PL=0
MOVL C00036 V=800.0 PL=0
MOVL C00037 V=800.0 PL=0
MOVL C00038 V=800.0 PL=0
MOVL C00039 V=800.0 PL=0
MOVL C00040 V=800.0 PL=0
MOVL C00041 V=800.0 PL=0
MOVL C00042 V=800.0 PL=0
MOVL C00043 V=800.0 PL=0
MOVL C00044 V=800.0 PL=0
MOVL C00045 V=800.0 PL=0
MOVL C00046 V=800.0 PL=0
MOVL C00047 V=800.0 PL=0
MOVL C00048 V=800.0 PL=0
MOVL C00049 V=800.0 PL=0
MOVL C00050 V=800.0 PL=0
MOVL C00051 V=800.0 PL=0
MOVL C00052 V=800.0 PL=0
MOVL C00053 V=800.0 PL=0
MOVL C00054 V=800.0 PL=0
MOVL C00055 V=800.0 PL=0
MOVL C00056 V=800.0 PL=0
MOVL C00057 V=800.0 PL=0
MOVL C00058 V=800.0 PL=0
MOVL C00059 V=800.0 PL=0
MOVL C00060 V=800.0 PL=0
MOVL C00061 V=800.0 PL=0
MOVL C00062 V=800.0 PL=0
MOVL C00063 V=800.0 PL=0
MOVL C00064 V=800.0 PL=0
MOVL C00065 V=800.0 PL=0
MOVL C00066 V=800.0 PL=0
MOVL C00067 V=800.0 PL=0
MOVL C00068 V=800.0 PL=0
MOVL C00069 V=800.0 PL=0
MOVL C00070 V=800.0 PL=0
MOVL C00071 V=800.0 PL=0
MOVL C00072 V=800.0 PL=0
MOVL C00073 V=800.0 PL=0
MOVL C00074 V=800.0 PL=0
MOVL C00075 V=800.0 PL=0
MOVL C00076 V=800.0 PL=0
MOVL C00077 V=800.0 PL=0
MOVL C00078 V=800.0 PL=0
MOVL C00079 V=800.0 PL=0
MOVL C00080 V=800.0 PL=0
MOVL C00081 V=800.0 PL=0
MOVL C00082 V=800.0 PL=0
MOVL C00083 V=800.0 PL=0
MOVL C00084 V=800.0 PL=0
MOVL C00085 V=800.0 PL=0
MOVL C00086 V=800.0 PL=0
MOVL C00087 V=800.0 PL=0
MOVL C00088 V=800.0 PL=0
MOVL C00089 V=800.0 PL=0
MOVL C00090 V=800.0 PL=0
MOVL C00091 V=800.0 PL=0
MOVL C00092 V=800.0 PL=0
MOVL C00093 V=800.0 PL=0
MOVL C00094 V=800.0 PL=0
MOVL C00095 V=800.0 PL=0
MOVL C00096 V=800.0 PL=0
MOVL C00097 V=800.0 PL=0
MOVL C00098 V=800.0 PL=0
MOVL C00099 V=800.0 PL=0
MOVL C00100 V=800.0 PL=0
MOVL C00101 V=800.0 PL=0
MOVL C00102 V=800.0 PL=0
MOVL C00103 V=800.0 PL=0
MOVL C00104 V=800.0 PL=0
MOVL C00105 V=800.0 PL=0
MOVL C00106 V=800.0 PL=0
MOVL C00107 V=800.0 PL=0
MOVL C00108 V=800.0 PL=0
MOVL C00109 V=800.0 PL=0
MOVL C00110 V=800.0 PL=0
MOVL C00111 V=800.0 PL=0
MOVL C00112 V=800.0 PL=0
MOVL C00113 V=800.0 PL=0
MOVL C00114 V=800.0 PL=0
MOVL C00115 V=800.0 PL=0
MOVL C00116 V=800.0 PL=0
MOVL C00117 V=800.0 PL=0
MOVL C00118 V=800.0 PL=0
MOVL C00119 V=800.0 PL=0
MOVL C00120 V=800.0 PL=0
MOVL C00121 V=800.0 PL=0
MOVL C00122 V=800.0 PL=0
MOVL C00123 V=800.0 PL=0
MOVL C00124 V=800.0 PL=0
MOVL C00125 V=800.0 PL=0
MOVL C00126 V=800.0 PL=0
MOVL C00127 V=800.0 PL=0
MOVL C00128 V=800.0 PL=0
MOVL C00129 V=800.0 PL=0
MOVL C00130 V=800.0 PL=0
MOVL C00131 V=800.0 PL=0
MOVL C00132 V=800.0 PL=0
MOVL C00133 V=800.0 PL=0
MOVL C00134 V=800.0 PL=0
MOVL C00135 V=800.0 PL=0
MOVL C00136 V=800.0 PL=0
MOVL C00137 V=800.0 PL=0
MOVL C00138 V=800.0 PL=0
MOVL C00139 V=800.0 PL=0
MOVL C00140 V=800.0 PL=0
MOVL C00141 V=800.0 PL=0
MOVL C00142 V=800.0 PL=0
MOVL C00143 V=800.0 PL=0
MOVL C00144 V=800.0 PL=0
MOVL C00145 V=800.0 PL=0
MOVL C00146 V=800.0 PL=0
MOVL C00147 V=800.0 PL=0
MOVL C00148 V=800.0 PL=0
MOVL C00149 V=800.0 PL=0
MOVL C00150 V=800.0 PL=0
MOVL C00151 V=800.0 PL=0
MOVL C00152 V=800.0 PL=0
MOVL C00153 V=800.0 PL=0
MOVL C00154 V=800.0 PL=0
MOVL C00155 V=800.0 PL=0
MOVL C00156 V=800.0 PL=0
MOVL C00157 V=800.0 PL=0
MOVL C00158 V=800.0 PL=0
MOVL C00159 V=800.0 PL=0
MOVL C00160 V=800.0 PL=0
MOVL C00161 V=800.0 PL=0
MOVL C00162 V=800.0 PL=0
MOVL C00163 V=800.0 PL=0
MOVL C00164 V=800.0 PL=0
MOVL C00165 V=800.0 PL=0
MOVL C00166 V=800.0 PL=0
MOVL C00167 V=800.0 PL=0
MOVL C00168 V=800.0 PL=0
MOVL C00169 V=800.0 PL=0
MOVL C00170 V=800.0 PL=0
MOVL C00171 V=800.0 PL=0
MOVL C00172 V=800.0 PL=0
MOVL C00173 V=800.0 PL=0
MOVL C00174 V=800.0 PL=0
MOVL C00175 V=800.0 PL=0
MOVL C00176 V=800.0 PL=0
MOVL C00177 V=800.0 PL=0
MOVL C00178 V=800.0 PL=0
MOVL C00179 V=800.0 PL=0
MOVL C00180 V=800.0 PL=0
MOVL C00181 V=800.0 PL=0
MOVL C00182 V=800.0 PL=0
MOVL C00183 V=800.0 PL=0
MOVL C00184 V=800.0 PL=0
MOVL C00185 V=800.0 PL=0
MOVL C00186 V=800.0 PL=0
MOVL C00187 V=800.0 PL=0
MOVL C00188 V=800.0 PL=0
MOVL C00189 V=800.0 PL=0
MOVL C00190 V=800.0 PL=0
MOVL C00191 V=800.0 PL=0
MOVL C00192 V=800.0 PL=0
MOVL C00193 V=800.0 PL=0
MOVL C00194 V=800.0 PL=0
MOVL C00195 V=800.0 PL=0
MOVL C00196 V=800.0 PL=0
MOVL C00197 V=800.0 PL=0
MOVL C00198 V=800.0 PL=0
MOVL C00199 V=800.0 PL=0
MOVL C00200 V=800.0 PL=0
MOVL C00201 V=800.0 PL=0
MOVL C00202 V=800.0 PL=0
MOVL C00203 V=800.0 PL=0
MOVL C00204 V=800.0 PL=0
MOVL C00205 V=800.0 PL=0
MOVL C00206 V=800.0 PL=0
MOVL C00207 V=800.0 PL=0
MOVL C00208 V=800.0 PL=0
MOVL C00209 V=800.0 PL=0
MOVL C00210 V=800.0 PL=0
MOVL C00211 V=800.0 PL=0
MOVL C00212 V=800.0 PL=0
MOVL C00213 V=800.0 PL=0
MOVL C00214 V=800.0 PL=0
MOVL C00215 V=800.0 PL=0
MOVL C00216 V=800.0 PL=0
MOVL C00217 V=800.0 PL=0
MOVL C00218 V=800.0 PL=0
MOVL C00219 V=800.0 PL=0
MOVL C00220 V=800.0 PL=0
MOVL C00221 V=800.0 PL=0
MOVL C00222 V=800.0 PL=0
MOVL C00223 V=800.0 PL=0
MOVL C00224 V=800.0 PL=0
MOVL C00225 V=800.0 PL=0
MOVL C00226 V=800.0 PL=0
MOVL C00227 V=800.0 PL=0
MOVL C00228 V=800.0 PL=0
MOVL C00229 V=800.0 PL=0
MOVL C00230 V=800.0 PL=0
MOVL C00231 V=800.0 PL=0
MOVL C00232 V=800.0 PL=0
MOVL C00233 V=800.0 PL=0
MOVL C00234 V=800.0 PL=0
MOVL C00235 V=800.0 PL=0
MOVL C00236 V=800.0 PL=0
MOVL C00237 V=800.0 PL=0
MOVL C00238 V=800.0 PL=0
MOVL C00239 V=800.0 PL=0
MOVL C00240 V=800.0 PL=0
MOVL C00241 V=800.0 PL=0
MOVL C00242 V=800.0 PL=0
MOVL C00243 V=800.0 PL=0
MOVL C00244 V=800.0 PL=0
MOVL C00245 V=800.0 PL=0
MOVL C00246 V=800.0 PL=0
MOVL C00247 V=800.0 PL=0
MOVL C00248 V=800.0 PL=0
MOVL C00249 V=800.0 PL=0
MOVL C00250 V=800.0 PL=0
MOVL C00251 V=800.0 PL=0
MOVL C00252 V=800.0 PL=0
MOVL C00253 V=800.0 PL=0
MOVL C00254 V=800.0 PL=0
MOVL C00255 V=800.0 PL=0
MOVL C00256 V=800.0 PL=0
MOVL C00257 V=800.0 PL=0
MOVL C00258 V=800.0 PL=0
MOVL C00259 V=800.0 PL=0
MOVL C00260 V=800.0 PL=0
MOVL C00261 V=800.0 PL=0
MOVL C00262 V=800.0 PL=0
MOVL C00263 V=800.0 PL=0
MOVL C00264 V=800.0 PL=0
MOVL C00265 V=800.0 PL=0
MOVL C00266 V=800.0 PL=0
MOVL C00267 V=800.0 PL=0
MOVL C00268 V=800.0 PL=0
MOVL C00269 V=800.0 PL=0
MOVL C00270 V=800.0 PL=0
MOVL C00271 V=800.0 PL=0
MOVL C00272 V=800.0 PL=0
MOVL C00273 V=800.0 PL=0
MOVL C00274 V=800.0 PL=0
MOVL C00275 V=800.0 PL=0
MOVL C00276 V=800.0 PL=0
MOVL C00277 V=800.0 PL=0
MOVL C00278 V=800.0 PL=0
MOVL C00279 V=800.0 PL=0
MOVL C00280 V=800.0 PL=0
MOVL C00281 V=800.0 PL=0
MOVL C00282 V=800.0 PL=0
MOVL C00283 V=800.0 PL=0
MOVL C00284 V=800.0 PL=0
MOVL C00285 V=800.0 PL=0
MOVL C00286 V=800.0 PL=0
MOVL C00287 V=800.0 PL=0
MOVL C00288 V=800.0 PL=0
MOVL C00289 V=800.0 PL=0
MOVL C00290 V=800.0 PL=0
MOVL C00291 V=800.0 PL=0
MOVL C00292 V=800.0 PL=0
MOVL C00293 V=800.0 PL=0
MOVL C00294 V=800.0 PL=0
MOVL C00295 V=800.0 PL=0
MOVL C00296 V=800.0 PL=0
MOVL C00297 V=800.0 PL=0
MOVL C00298 V=800.0 PL=0
MOVL C00299 V=800.0 PL=0
MOVL C00300 V=800.0 PL=0
MOVL C00301 V=800.0 PL=0
MOVL C00302 V=800.0 PL=0
MOVL C00303 V=800.0 PL=0
MOVL C00304 V=800.0 PL=0
MOVL C00305 V=800.0 PL=0
MOVL C00306 V=800.0 PL=0
MOVL C00307 V=800.0 PL=0
MOVL C00308 V=800.0 PL=0
MOVL C00309 V=800.0 PL=0
MOVL C00310 V=800.0 PL=0
MOVL C00311 V=800.0 PL=0
MOVL C00312 V=800.0 PL=0
MOVL C00313 V=800.0 PL=0
MOVL C00314 V=800.0 PL=0
MOVL C00315 V=800.0 PL=0
MOVL C00316 V=800.0 PL=0
MOVL C00317 V=800.0 PL=0
MOVL C00318 V=800.0 PL=0
MOVL C00319 V=800.0 PL=0
MOVL C00320 V=800.0 PL=0
MOVL C00321 V=800.0 PL=0
MOVL C00322 V=800.0 PL=0
MOVL C00323 V=800.0 PL=0
MOVL C00324 V=800.0 PL=0
MOVL C00325 V=800.0 PL=0
MOVL C00326 V=800.0 PL=0
MOVL C00327 V=800.0 PL=0
MOVL C00328 V=800.0 PL=0
MOVL C00329 V=800.0 PL=0
MOVL C00330 V=800.0 PL=0
MOVL C00331 V=800.0 PL=0
MOVL C00332 V=800.0 PL=0
MOVL C00333 V=800.0 PL=0
MOVL C00334 V=800.0 PL=0
MOVL C00335 V=800.0 PL=0
MOVL C00336 V=800.0 PL=0
MOVL C00337 V=800.0 PL=0
MOVL C00338 V=800.0 PL=0
MOVL C00339 V=800.0 PL=0
MOVL C00340 V=800.0 PL=0
MOVL C00341 V=800.0 PL=0
MOVL C00342 V=800.0 PL=0
MOVL C00343 V=800.0 PL=0
MOVL C00344 V=800.0 PL=0
MOVL C00345 V=800.0 PL=0
MOVL C00346 V=800.0 PL=0
MOVL C00347 V=800.0 PL=0
MOVL C00348 V=800.0 PL=0
MOVL C00349 V=800.0 PL=0
MOVL C00350 V=800.0 PL=0
MOVL C00351 V=800.0 PL=0
MOVL C00352 V=800.0 PL=0
MOVL C00353 V=800.0 PL=0
MOVL C00354 V=800.0 PL=0
MOVL C00355 V=800.0 PL=0
MOVL C00356 V=800.0 PL=0
MOVL C00357 V=800.0 PL=0
MOVL C00358 V=800.0 PL=0
MOVL C00359 V=800.0 PL=0
MOVL C00360 V=800.0 PL=0
MOVL C00361 V=800.0 PL=0
MOVL C00362 V=800.0 PL=0
MOVL C00363 V=800.0 PL=0
MOVL C00364 V=800.0 PL=0
MOVL C00365 V=800.0 PL=0
MOVL C00366 V=800.0 PL=0
MOVL C00367 V=800.0 PL=0
MOVL C00368 V=800.0 PL=0
MOVL C00369 V=800.0 PL=0
MOVL C00370 V=800.0 PL=0
MOVL C00371 V=800.0 PL=0
MOVL C00372 V=800.0 PL=0
MOVL C00373 V=800.0 PL=0
MOVL C00374 V=800.0 PL=0
MOVL C00375 V=800.0 PL=0
MOVL C00376 V=800.0 PL=0
MOVL C00377 V=800.0 PL=0
MOVL C00378 V=800.0 PL=0
MOVL C00379 V=800.0 PL=0
MOVL C00380 V=800.0 PL=0
MOVL C00381 V=800.0 PL=0
MOVL C00382 V=800.0 PL=0
MOVL C00383 V=800.0 PL=0
MOVL C00384 V=800.0 PL=0
MOVL C00385 V=800.0 PL=0
MOVL C00386 V=800.0 PL=0
MOVL C00387 V=800.0 PL=0
MOVL C00388 V=800.0 PL=0
MOVL C00389 V=800.0 PL=0
MOVL C00390 V=800.0 PL=0
MOVL C00391 V=800.0 PL=0
MOVL C00392 V=800.0 PL=0
MOVL C00393 V=800.0 PL=0
MOVL C00394 V=800.0 PL=0
MOVL C00395 V=800.0 PL=0
MOVL C00396 V=800.0 PL=0
MOVL C00397 V=800.0 PL=0
MOVL C00398 V=800.0 PL=0
MOVL C00399 V=800.0 PL=0
MOVL C00400 V=800.0 PL=0
MOVL C00401 V=800.0 PL=0
MOVL C00402 V=800.0 PL=0
MOVL C00403 V=800.0 PL=0
MOVL C00404 V=800.0 PL=0
MOVL C00405 V=800.0 PL=0
MOVL C00406 V=800.0 PL=0
MOVL C00407 V=800.0 PL=0
MOVL C00408 V=800.0 PL=0
MOVL C00409 V=800.0 PL=0
MOVL C00410 V=800.0 PL=0
MOVL C00411 V=800.0 PL=0
MOVL C00412 V=800.0 PL=0
MOVL C00413 V=800.0 PL=0
MOVL C00414 V=800.0 PL=0
MOVL C00415 V=800.0 PL=0
MOVL C00416 V=800.0 PL=0
MOVL C00417 V=800.0 PL=0
MOVL C00418 V=800.0 PL=0
MOVL C00419 V=800.0 PL=0
MOVL C00420 V=800.0 PL=0
MOVL C00421 V=800.0 PL=0
MOVL C00422 V=800.0 PL=0
MOVL C00423 V=800.0 PL=0
MOVL C00424 V=800.0 PL=0
MOVL C00425 V=800.0 PL=0
MOVL C00426 V=800.0 PL=0
MOVL C00427 V=800.0 PL=0
MOVL C00428 V=800.0 PL=0
MOVL C00429 V=800.0 PL=0
MOVL C00430 V=800.0 PL=0
MOVL C00431 V=800.0 PL=0
MOVL C00432 V=800.0 PL=0
MOVL C00433 V=800.0 PL=0
MOVL C00434 V=800.0 PL=0
MOVL C00435 V=800.0 PL=0
MOVL C00436 V=800.0 PL=0
MOVL C00437 V=800.0 PL=0
MOVL C00438 V=800.0 PL=0
MOVL C00439 V=800.0 PL=0
MOVL C00440 V=800.0 PL=0
MOVL C00441 V=800.0 PL=0
MOVL C00442 V=800.0 PL=0
MOVL C00443 V=800.0 PL=0
MOVL C00444 V=800.0 PL=0
MOVL C00445 V=800.0 PL=0
MOVL C00446 V=800.0 PL=0
MOVL C00447 V=800.0 PL=0
MOVL C00448 V=800.0 PL=0
MOVL C00449 V=800.0 PL=0
MOVL C00450 V=800.0 PL=0
MOVL C00451 V=800.0 PL=0
MOVL C00452 V=800.0 PL=0
MOVL C00453 V=800.0 PL=0
MOVL C00454 V=800.0 PL=0
MOVL C00455 V=800.0 PL=0
MOVL C00456 V=800.0 PL=0
MOVL C00457 V=800.0 PL=0
MOVL C00458 V=800.0 PL=0
MOVL C00459 V=800.0 PL=0
MOVL C00460 V=800.0 PL=0
MOVL C00461 V=800.0 PL=0
MOVL C00462 V=800.0 PL=0
MOVL C00463 V=800.0 PL=0
MOVL C00464 V=800.0 PL=0
MOVL C00465 V=800.0 PL=0
MOVL C00466 V=800.0 PL=0
MOVL C00467 V=800.0 PL=0
MOVL C00468 V=800.0 PL=0
MOVL C00469 V=800.0 PL=0
MOVL C00470 V=800.0 PL=0
MOVL C00471 V=800.0 PL=0
MOVL C00472 V=800.0 PL=0
MOVL C00473 V=800.0 PL=0
MOVL C00474 V=800.0 PL=0
MOVL C00475 V=800.0 PL=0
MOVL C00476 V=800.0 PL=0
MOVL C00477 V=800.0 PL=0
MOVL C00478 V=800.0 PL=0
MOVL C00479 V=800.0 PL=0
MOVL C00480 V=800.0 PL=0
MOVL C00481 V=800.0 PL=0
MOVL C00482 V=800.0 PL=0
MOVL C00483 V=800.0 PL=0
MOVL C00484 V=800.0 PL=0
MOVL C00485 V=800.0 PL=0
MOVL C00486 V=800.0 PL=0
MOVL C00487 V=800.0 PL=0
MOVL C00488 V=800.0 PL=0
MOVL C00489 V=800.0 PL=0
MOVL C00490 V=800.0 PL=0
MOVL C00491 V=800.0 PL=0
MOVL C00492 V=800.0 PL=0
MOVL C00493 V=800.0 PL=0
MOVL C00494 V=800.0 PL=0
MOVL C00495 V=800.0 PL=0
MOVL C00496 V=800.0 PL=0
MOVL C00497 V=800.0 PL=0
MOVL C00498 V=800.0 PL=0
MOVL C00499 V=800.0 PL=0
MOVL C00500 V=800.0 PL=0
MOVL C00501 V=800.0 PL=0
MOVL C00502 V=800.0 PL=0
MOVL C00503 V=800.0 PL=0
MOVL C00504 V=800.0 PL=0
MOVL C00505 V=800.0 PL=0
MOVL C00506 V=800.0 PL=0
MOVL C00507 V=800.0 PL=0
MOVL C00508 V=800.0 PL=0
MOVL C00509 V=800.0 PL=0
MOVL C00510 V=800.0 PL=0
MOVL C00511 V=800.0 PL=0
MOVL C00512 V=800.0 PL=0
MOVL C00513 V=800.0 PL=0
MOVL C00514 V=800.0 PL=0
MOVL C00515 V=800.0 PL=0
MOVL C00516 V=800.0 PL=0
MOVL C00517 V=800.0 PL=0
MOVL C00518 V=800.0 PL=0
MOVL C00519 V=800.0 PL=0
MOVL C00520 V=800.0 PL=0
MOVL C00521 V=800.0 PL=0
MOVL C00522 V=800.0 PL=0
MOVL C00523 V=800.0 PL=0
MOVL C00524 V=800.0 PL=0
MOVL C00525 V=800.0 PL=0
MOVL C00526 V=800.0 PL=0
MOVL C00527 V=800.0 PL=0
MOVL C00528 V=800.0 PL=0
MOVL C00529 V=800.0 PL=0
MOVL C00530 V=800.0 PL=0
MOVL C00531 V=800.0 PL=0
MOVL C00532 V=800.0 PL=0
MOVL C00533 V=800.0 PL=0
MOVL C00534 V=800.0 PL=0
MOVL C00535 V=800.0 PL=0
MOVL C00536 V=800.0 PL=0
MOVL C00537 V=800.0 PL=0
MOVL C00538 V=800.0 PL=0
MOVL C00539 V=800.0 PL=0
MOVL C00540 V=800.0 PL=0
MOVL C00541 V=800.0 PL=0
MOVL C00542 V=800.0 PL=0
MOVL C00543 V=800.0 PL=0
MOVL C00544 V=800.0 PL=0
MOVL C00545 V=800.0 PL=0
MOVL C00546 V=800.0 PL=0
MOVL C00547 V=800.0 PL=0
MOVL C00548 V=800.0 PL=0
MOVL C00549 V=800.0 PL=0
MOVL C00550 V=800.0 PL=0
MOVL C00551 V=800.0 PL=0
MOVL C00552 V=800.0 PL=0
MOVL C00553 V=800.0 PL=0
MOVL C00554 V=800.0 PL=0
MOVL C00555 V=800.0 PL=0
MOVL C00556 V=800.0 PL=0
MOVL C00557 V=800.0 PL=0
MOVL C00558 V=800.0 PL=0
MOVL C00559 V=800.0 PL=0
MOVL C00560 V=800.0 PL=0
MOVL C00561 V=800.0 PL=0
MOVL C00562 V=800.0 PL=0
MOVL C00563 V=800.0 PL=0
MOVL C00564 V=800.0 PL=0
MOVL C00565 V=800.0 PL=0
MOVL C00566 V=800.0 PL=0
MOVL C00567 V=800.0 PL=0
MOVL C00568 V=800.0 PL=0
MOVL C00569 V=800.0 PL=0
MOVL C00570 V=800.0 PL=0
MOVL C00571 V=800.0 PL=0
MOVL C00572 V=800.0 PL=0
MOVL C00573 V=800.0 PL=0
MOVL C00574 V=800.0 PL=0
MOVL C00575 V=800.0 PL=0
MOVL C00576 V=800.0 PL=0
MOVL C00577 V=800.0 PL=0
MOVL C00578 V=800.0 PL=0
MOVL C00579 V=800.0 PL=0
MOVL C00580 V=800.0 PL=0
MOVL C00581 V=800.0 PL=0
MOVL C00582 V=800.0 PL=0
MOVL C00583 V=800.0 PL=0
MOVL C00584 V=800.0 PL=0
MOVL C00585 V=800.0 PL=0
MOVL C00586 V=800.0 PL=0
MOVL C00587 V=800.0 PL=0
MOVL C00588 V=800.0 PL=0
MOVL C00589 V=800.0 PL=0
MOVL C00590 V=800.0 PL=0
MOVL C00591 V=800.0 PL=0
MOVL C00592 V=800.0 PL=0
MOVL C00593 V=800.0 PL=0
MOVL C00594 V=800.0 PL=0
MOVL C00595 V=800.0 PL=0
MOVL C00596 V=800.0 PL=0
MOVL C00597 V=800.0 PL=0
MOVL C00598 V=800.0 PL=0
MOVL C00599 V=800.0 PL=0
MOVL C00600 V=800.0 PL=0
MOVL C00601 V=800.0 PL=0
MOVL C00602 V=800.0 PL=0
MOVL C00603 V=800.0 PL=0
MOVL C00604 V=800.0 PL=0
MOVL C00605 V=800.0 PL=0
MOVL C00606 V=800.0 PL=0
MOVL C00607 V=800.0 PL=0
MOVL C00608 V=800.0 PL=0
MOVL C00609 V=800.0 PL=0
MOVL C00610 V=800.0 PL=0
MOVL C00611 V=800.0 PL=0
MOVL C00612 V=800.0 PL=0
MOVL C00613 V=800.0 PL=0
MOVL C00614 V=800.0 PL=0
MOVL C00615 V=800.0 PL=0
MOVL C00616 V=800.0 PL=0
MOVL C00617 V=800.0 PL=0
MOVL C00618 V=800.0 PL=0
MOVL C00619 V=800.0 PL=0
MOVL C00620 V=800.0 PL=0
MOVL C00621 V=800.0 PL=0
MOVL C00622 V=800.0 PL=0
MOVL C00623 V=800.0 PL=0
MOVL C00624 V=800.0 PL=0
MOVL C00625 V=800.0 PL=0
MOVL C00626 V=800.0 PL=0
MOVL C00627 V=800.0 PL=0
MOVL C00628 V=800.0 PL=0
MOVL C00629 V=800.0 PL=0
MOVL C00630 V=800.0 PL=0
MOVL C00631 V=800.0 PL=0
MOVL C00632 V=800.0 PL=0
MOVL C00633 V=800.0 PL=0
MOVL C00634 V=800.0 PL=0
MOVL C00635 V=800.0 PL=0
MOVL C00636 V=800.0 PL=0
MOVL C00637 V=800.0 PL=0
MOVL C00638 V=800.0 PL=0
MOVL C00639 V=800.0 PL=0
MOVL C00640 V=800.0 PL=0
MOVL C00641 V=800.0 PL=0
MOVL C00642 V=800.0 PL=0
MOVL C00643 V=800.0 PL=0
MOVL C00644 V=800.0 PL=0
MOVL C00645 V=800.0 PL=0
MOVL C00646 V=800.0 PL=0
MOVL C00647 V=800.0 PL=0
MOVL C00648 V=800.0 PL=0
MOVL C00649 V=800.0 PL=0
MOVL C00650 V=800.0 PL=0
MOVL C00651 V=800.0 PL=0
MOVL C00652 V=800.0 PL=0
MOVL C00653 V=800.0 PL=0
MOVL C00654 V=800.0 PL=0
MOVL C00655 V=800.0 PL=0
MOVL C00656 V=800.0 PL=0
MOVL C00657 V=800.0 PL=0
MOVL C00658 V=800.0 PL=0
MOVL C00659 V=800.0 PL=0
MOVL C00660 V=800.0 PL=0
MOVL C00661 V=800.0 PL=0
MOVL C00662 V=800.0 PL=0
MOVL C00663 V=800.0 PL=0
MOVL C00664 V=800.0 PL=0
MOVL C00665 V=800.0 PL=0
MOVL C00666 V=800.0 PL=0
MOVL C00667 V=800.0 PL=0
MOVL C00668 V=800.0 PL=0
MOVL C00669 V=800.0 PL=0
MOVL C00670 V=800.0 PL=0
MOVL C00671 V=800.0 PL=0
MOVL C00672 V=800.0 PL=0
MOVL C00673 V=800.0 PL=0
MOVL C00674 V=800.0 PL=0
MOVL C00675 V=800.0 PL=0
MOVL C00676 V=800.0 PL=0
MOVL C00677 V=800.0 PL=0
MOVL C00678 V=800.0 PL=0
MOVL C00679 V=800.0 PL=0
MOVL C00680 V=800.0 PL=0
MOVL C00681 V=800.0 PL=0
MOVL C00682 V=800.0 PL=0
MOVL C00683 V=800.0 PL=0
MOVL C00684 V=800.0 PL=0
MOVL C00685 V=800.0 PL=0
MOVL C00686 V=800.0 PL=0
MOVL C00687 V=800.0 PL=0
MOVL C00688 V=800.0 PL=0
MOVL C00689 V=800.0 PL=0
MOVL C00690 V=800.0 PL=0
MOVL C00691 V=800.0 PL=0
MOVL C00692 V=800.0 PL=0
MOVL C00693 V=800.0 PL=0
MOVL C00694 V=800.0 PL=0
MOVL C00695 V=800.0 PL=0
MOVL C00696 V=800.0 PL=0
MOVL C00697 V=800.0 PL=0
MOVL C00698 V=800.0 PL=0
MOVL C00699 V=800.0 PL=0
MOVL C00700 V=800.0 PL=0
MOVL C00701 V=800.0 PL=0
MOVL C00702 V=800.0 PL=0
MOVL C00703 V=800.0 PL=0
MOVL C00704 V=800.0 PL=0
MOVL C00705 V=800.0 PL=0
MOVL C00706 V=800.0 PL=0
MOVL C00707 V=800.0 PL=0
MOVL C00708 V=800.0 PL=0
MOVL C00709 V=800.0 PL=0
MOVL C00710 V=800.0 PL=0
MOVL C00711 V=800.0 PL=0
MOVL C00712 V=800.0 PL=0
MOVL C00713 V=800.0 PL=0
MOVL C00714 V=800.0 PL=0
MOVL C00715 V=800.0 PL=0
MOVL C00716 V=800.0 PL=0
MOVL C00717 V=800.0 PL=0
MOVL C00718 V=800.0 PL=0
MOVL C00719 V=800.0 PL=0
MOVL C00720 V=800.0 PL=0
MOVL C00721 V=800.0 PL=0
MOVL C00722 V=800.0 PL=0
MOVL C00723 V=800.0 PL=0
MOVL C00724 V=800.0 PL=0
MOVL C00725 V=800.0 PL=0
MOVL C00726 V=800.0 PL=0
MOVL C00727 V=800.0 PL=0
MOVL C00728 V=800.0 PL=0
MOVL C00729 V=800.0 PL=0
MOVL C00730 V=800.0 PL=0
MOVL C00731 V=800.0 PL=0
MOVL C00732 V=800.0 PL=0
MOVL C00733 V=800.0 PL=0
MOVL C00734 V=800.0 PL=0
MOVL C00735 V=800.0 PL=0
MOVL C00736 V=800.0 PL=0
MOVL C00737 V=800.0 PL=0
MOVL C00738 V=800.0 PL=0
MOVL C00739 V=800.0 PL=0
MOVL C00740 V=800.0 PL=0
MOVL C00741 V=800.0 PL=0
MOVL C00742 V=800.0 PL=0
MOVL C00743 V=800.0 PL=0
MOVL C00744 V=800.0 PL=0
MOVL C00745 V=800.0 PL=0
MOVL C00746 V=800.0 PL=0
MOVL C00747 V=800.0 PL=0
MOVL C00748 V=800.0 PL=0
MOVL C00749 V=800.0 PL=0
MOVL C00750 V=800.0 PL=0
MOVL C00751 V=800.0 PL=0
MOVL C00752 V=800.0 PL=0
MOVL C00753 V=800.0 PL=0
MOVL C00754 V=800.0 PL=0
MOVL C00755 V=800.0 PL=0
MOVL C00756 V=800.0 PL=0
MOVL C00757 V=800.0 PL=0
MOVL C00758 V=800.0 PL=0
MOVL C00759 V=800.0 PL=0
MOVL C00760 V=800.0 PL=0
MOVL C00761 V=800.0 PL=0
MOVL C00762 V=800.0 PL=0
MOVL C00763 V=800.0 PL=0
MOVL C00764 V=800.0 PL=0
MOVL C00765 V=800.0 PL=0
MOVL C00766 V=800.0 PL=0
MOVL C00767 V=800.0 PL=0
MOVL C00768 V=800.0 PL=0
MOVL C00769 V=800.0 PL=0
MOVL C00770 V=800.0 PL=0
MOVL C00771 V=800.0 PL=0
MOVL C00772 V=800.0 PL=0
MOVL C00773 V=800.0 PL=0
MOVL C00774 V=800.0 PL=0
MOVL C00775 V=800.0 PL=0
MOVL C00776 V=800.0 PL=0
MOVL C00777 V=800.0 PL=0
MOVL C00778 V=800.0 PL=0
MOVL C00779 V=800.0 PL=0
MOVL C00780 V=800.0 PL=0
MOVL C00781 V=800.0 PL=0
MOVL C00782 V=800.0 PL=0
MOVL C00783 V=800.0 PL=0
MOVL C00784 V=800.0 PL=0
MOVL C00785 V=800.0 PL=0
MOVL C00786 V=800.0 PL=0
MOVL C00787 V=800.0 PL=0
MOVL C00788 V=800.0 PL=0
MOVL C00789 V=800.0 PL=0
MOVL C00790 V=800.0 PL=0
MOVL C00791 V=800.0 PL=0
MOVL C00792 V=800.0 PL=0
MOVL C00793 V=800.0 PL=0
MOVL C00794 V=800.0 PL=0
MOVL C00795 V=800.0 PL=0
MOVL C00796 V=800.0 PL=0
MOVL C00797 V=800.0 PL=0
MOVL C00798 V=800.0 PL=0
MOVL C00799 V=800.0 PL=0
MOVL C00800 V=800.0 PL=0
MOVL C00801 V=800.0 PL=0
MOVL C00802 V=800.0 PL=0
MOVL C00803 V=800.0 PL=0
MOVL C00804 V=800.0 PL=0
MOVL C00805 V=800.0 PL=0
MOVL C00806 V=800.0 PL=0
MOVL C00807 V=800.0 PL=0
MOVL C00808 V=800.0 PL=0
MOVL C00809 V=800.0 PL=0
MOVL C00810 V=800.0 PL=0
MOVL C00811 V=800.0 PL=0
MOVL C00812 V=800.0 PL=0
MOVL C00813 V=800.0 PL=0
MOVL C00814 V=800.0 PL=0
MOVL C00815 V=800.0 PL=0
MOVL C00816 V=800.0 PL=0
MOVL C00817 V=800.0 PL=0
MOVL C00818 V=800.0 PL=0
MOVL C00819 V=800.0 PL=0
MOVL C00820 V=800.0 PL=0
MOVL C00821 V=800.0 PL=0
MOVL C00822 V=800.0 PL=0
MOVL C00823 V=800.0 PL=0
MOVL C00824 V=800.0 PL=0
MOVL C00825 V=800.0 PL=0
MOVL C00826 V=800.0 PL=0
MOVL C00827 V=800.0 PL=0
MOVL C00828 V=800.0 PL=0
MOVL C00829 V=800.0 PL=0
MOVL C00830 V=800.0 PL=0
MOVL C00831 V=800.0 PL=0
MOVL C00832 V=800.0 PL=0
MOVL C00833 V=800.0 PL=0
MOVL C00834 V=800.0 PL=0
MOVL C00835 V=800.0 PL=0
MOVL C00836 V=800.0 PL=0
MOVL C00837 V=800.0 PL=0
MOVL C00838 V=800.0 PL=0
MOVL C00839 V=800.0 PL=0
MOVL C00840 V=800.0 PL=0
MOVL C00841 V=800.0 PL=0
MOVL C00842 V=800.0 PL=0
MOVL C00843 V=800.0 PL=0
MOVL C00844 V=800.0 PL=0
MOVL C00845 V=800.0 PL=0
MOVL C00846 V=800.0 PL=0
MOVL C00847 V=800.0 PL=0
MOVL C00848 V=800.0 PL=0
MOVL C00849 V=800.0 PL=0
MOVL C00850 V=800.0 PL=0
MOVL C00851 V=800.0 PL=0
MOVL C00852 V=800.0 PL=0
MOVL C00853 V=800.0 PL=0
MOVL C00854 V=800.0 PL=0
MOVL C00855 V=800.0 PL=0
MOVL C00856 V=800.0 PL=0
MOVL C00857 V=800.0 PL=0
MOVL C00858 V=800.0 PL=0
MOVL C00859 V=800.0 PL=0
MOVL C00860 V=800.0 PL=0
MOVL C00861 V=800.0 PL=0
MOVL C00862 V=800.0 PL=0
MOVL C00863 V=800.0 PL=0
MOVL C00864 V=800.0 PL=0
MOVL C00865 V=800.0 PL=0
MOVL C00866 V=800.0 PL=0
MOVL C00867 V=800.0 PL=0
MOVL C00868 V=800.0 PL=0
MOVL C00869 V=800.0 PL=0
MOVL C00870 V=800.0 PL=0
MOVL C00871 V=800.0 PL=0
MOVL C00872 V=800.0 PL=0
MOVL C00873 V=800.0 PL=0
MOVL C00874 V=800.0 PL=0
MOVL C00875 V=800.0 PL=0
MOVL C00876 V=800.0 PL=0
MOVL C00877 V=800.0 PL=0
MOVL C00878 V=800.0 PL=0
MOVL C00879 V=800.0 PL=0
MOVL C00880 V=800.0 PL=0
MOVL C00881 V=800.0 PL=0
MOVL C00882 V=800.0 PL=0
MOVL C00883 V=800.0 PL=0
MOVL C00884 V=800.0 PL=0
MOVL C00885 V=800.0 PL=0
MOVL C00886 V=800.0 PL=0
MOVL C00887 V=800.0 PL=0
MOVL C00888 V=800.0 PL=0
MOVL C00889 V=800.0 PL=0
MOVL C00890 V=800.0 PL=0
MOVL C00891 V=800.0 PL=0
MOVL C00892 V=800.0 PL=0
MOVL C00893 V=800.0 PL=0
MOVL C00894 V=800.0 PL=0
MOVL C00895 V=800.0 PL=0
MOVL C00896 V=800.0 PL=0
MOVL C00897 V=800.0 PL=0
MOVL C00898 V=800.0 PL=0
MOVL C00899 V=800.0 PL=0
MOVL C00900 V=800.0 PL=0
MOVL C00901 V=800.0 PL=0
MOVL C00902 V=800.0 PL=0
MOVL C00903 V=800.0 PL=0
MOVL C00904 V=800.0 PL=0
MOVL C00905 V=800.0 PL=0
MOVL C00906 V=800.0 PL=0
MOVL C00907 V=800.0 PL=0
MOVL C00908 V=800.0 PL=0
MOVL C00909 V=800.0 PL=0
MOVL C00910 V=800.0 PL=0
MOVL C00911 V=800.0 PL=0
MOVL C00912 V=800.0 PL=0
MOVL C00913 V=800.0 PL=0
MOVL C00914 V=800.0 PL=0
MOVL C00915 V=800.0 PL=0
MOVL C00916 V=800.0 PL=0
MOVL C00917 V=800.0 PL=0
MOVL C00918 V=800.0 PL=0
MOVL C00919 V=800.0 PL=0
MOVL C00920 V=800.0 PL=0
MOVL C00921 V=800.0 PL=0
MOVL C00922 V=800.0 PL=0
MOVL C00923 V=800.0 PL=0
MOVL C00924 V=800.0 PL=0
MOVL C00925 V=800.0 PL=0
MOVL C00926 V=800.0 PL=0
MOVL C00927 V=800.0 PL=0
MOVL C00928 V=800.0 PL=0
MOVL C00929 V=800.0 PL=0
MOVL C00930 V=800.0 PL=0
MOVL C00931 V=800.0 PL=0
MOVL C00932 V=800.0 PL=0
MOVL C00933 V=800.0 PL=0
MOVL C00934 V=800.0 PL=0
MOVL C00935 V=800.0 PL=0
MOVL C00936 V=800.0 PL=0
MOVL C00937 V=800.0 PL=0
MOVL C00938 V=800.0 PL=0
MOVL C00939 V=800.0 PL=0
MOVL C00940 V=800.0 PL=0
MOVL C00941 V=800.0 PL=0
MOVL C00942 V=800.0 PL=0
MOVL C00943 V=800.0 PL=0
MOVL C00944 V=800.0 PL=0
MOVL C00945 V=800.0 PL=0
MOVL C00946 V=800.0 PL=0
MOVL C00947 V=800.0 PL=0
MOVL C00948 V=800.0 PL=0
MOVL C00949 V=800.0 PL=0
MOVL C00950 V=800.0 PL=0
MOVL C00951 V=800.0 PL=0
MOVL C00952 V=800.0 PL=0
MOVL C00953 V=800.0 PL=0
MOVL C00954 V=800.0 PL=0
MOVL C00955 V=800.0 PL=0
MOVL C00956 V=800.0 PL=0
MOVL C00957 V=800.0 PL=0
MOVL C00958 V=800.0 PL=0
MOVL C00959 V=800.0 PL=0
MOVL C00960 V=800.0 PL=0
MOVL C00961 V=800.0 PL=0
MOVL C00962 V=800.0 PL=0
MOVL C00963 V=800.0 PL=0
MOVL C00964 V=800.0 PL=0
MOVL C00965 V=800.0 PL=0
MOVL C00966 V=800.0 PL=0
MOVL C00967 V=800.0 PL=0
MOVL C00968 V=800.0 PL=0
MOVL C00969 V=800.0 PL=0
MOVL C00970 V=800.0 PL=0
MOVL C00971 V=800.0 PL=0
MOVL C00972 V=800.0 PL=0
MOVL C00973 V=800.0 PL=0
MOVL C00974 V=800.0 PL=0
MOVL C00975 V=800.0 PL=0
MOVL C00976 V=800.0 PL=0
MOVL C00977 V=800.0 PL=0
MOVL C00978 V=800.0 PL=0
MOVL C00979 V=800.0 PL=0
MOVL C00980 V=800.0 PL=0
MOVL C00981 V=800.0 PL=0
MOVL C00982 V=800.0 PL=0
MOVL C00983 V=800.0 PL=0
MOVL C00984 V=800.0 PL=0
MOVL C00985 V=800.0 PL=0
MOVL C00986 V=800.0 PL=0
MOVL C00987 V=800.0 PL=0
MOVL C00988 V=800.0 PL=0
MOVL C00989 V=800.0 PL=0
MOVL C00990 V=800.0 PL=0
MOVL C00991 V=800.0 PL=0
MOVL C00992 V=800.0 PL=0
MOVL C00993 V=800.0 PL=0
MOVL C00994 V=800.0 PL=0
MOVL C00995 V=800.0 PL=0
MOVL C00996 V=800.0 PL=0
MOVL C00997 V=800.0 PL=0
MOVL C00998 V=800.0 PL=0
MOVL C00999 V=800.0 PL=0
MOVL C01000 V=800.0 PL=0
MOVL C01001 V=800.0 PL=0
MOVL C01002 V=800.0 PL=0
MOVL C01003 V=800.0 PL=0
MOVL C01004 V=800.0 PL=0
MOVL C01005 V=800.0 PL=0
MOVL C01006 V=800.0 PL=0
MOVL C01007 V=800.0 PL=0
MOVL C01008 V=800.0 PL=0
MOVL C01009 V=800.0 PL=0
MOVL C01010 V=800.0 PL=0
MOVL C01011 V=800.0 PL=0
MOVL C01012 V=800.0 PL=0
MOVL C01013 V=800.0 PL=0
MOVL C01014 V=800.0 PL=0
MOVL C01015 V=800.0 PL=0
MOVL C01016 V=800.0 PL=0
MOVL C01017 V=800.0 PL=0
MOVL C01018 V=800.0 PL=0
MOVL C01019 V=800.0 PL=0
MOVL C01020 V=800.0 PL=0
MOVL C01021 V=800.0 PL=0
MOVL C01022 V=800.0 PL=0
MOVL C01023 V=800.0 PL=0
MOVL C01024 V=800.0 PL=0
MOVL C01025 V=800.0 PL=0
MOVL C01026 V=800.0 PL=0
MOVL C01027 V=800.0 PL=0
MOVL C01028 V=800.0 PL=0
MOVL C01029 V=800.0 PL=0
MOVL C01030 V=800.0 PL=0
MOVL C01031 V=800.0 PL=0
MOVL C01032 V=800.0 PL=0
MOVL C01033 V=800.0 PL=0
MOVL C01034 V=800.0 PL=0
MOVL C01035 V=800.0 PL=0
MOVL C01036 V=800.0 PL=0
MOVL C01037 V=800.0 PL=0
MOVL C01038 V=800.0 PL=0
MOVL C01039 V=800.0 PL=0
MOVL C01040 V=800.0 PL=0
MOVL C01041 V=800.0 PL=0
MOVL C01042 V=800.0 PL=0
MOVL C01043 V=800.0 PL=0
MOVL C01044 V=800.0 PL=0
MOVL C01045 V=800.0 PL=0
MOVL C01046 V=800.0 PL=0
MOVL C01047 V=800.0 PL=0
MOVL C01048 V=800.0 PL=0
MOVL C01049 V=800.0 PL=0
MOVL C01050 V=800.0 PL=0
MOVL C01051 V=800.0 PL=0
MOVL C01052 V=800.0 PL=0
MOVL C01053 V=800.0 PL=0
MOVL C01054 V=800.0 PL=0
MOVL C01055 V=800.0 PL=0
MOVL C01056 V=800.0 PL=0
MOVL C01057 V=800.0 PL=0
MOVL C01058 V=800.0 PL=0
MOVL C01059 V=800.0 PL=0
MOVL C01060 V=800.0 PL=0
MOVL C01061 V=800.0 PL=0
MOVL C01062 V=800.0 PL=0
MOVL C01063 V=800.0 PL=0
MOVL C01064 V=800.0 PL=0
MOVL C01065 V=800.0 PL=0
MOVL C01066 V=800.0 PL=0
MOVL C01067 V=800.0 PL=0
MOVL C01068 V=800.0 PL=0
MOVL C01069 V=800.0 PL=0
MOVL C01070 V=800.0 PL=0
MOVL C01071 V=800.0 PL=0
MOVL C01072 V=800.0 PL=0
MOVL C01073 V=800.0 PL=0
MOVL C01074 V=800.0 PL=0
MOVL C01075 V=800.0 PL=0
MOVL C01076 V=800.0 PL=0
MOVL C01077 V=800.0 PL=0
MOVL C01078 V=800.0 PL=0
MOVL C01079 V=800.0 PL=0
MOVL C01080 V=800.0 PL=0
MOVL C01081 V=800.0 PL=0
MOVL C01082 V=800.0 PL=0
MOVL C01083 V=800.0 PL=0
MOVL C01084 V=800.0 PL=0
MOVL C01085 V=800.0 PL=0
MOVL C01086 V=800.0 PL=0
MOVL C01087 V=800.0 PL=0
MOVL C01088 V=800.0 PL=0
MOVL C01089 V=800.0 PL=0
MOVL C01090 V=800.0 PL=0
MOVL C01091 V=800.0 PL=0
MOVL C01092 V=800.0 PL=0
MOVL C01093 V=800.0 PL=0
MOVL C01094 V=800.0 PL=0
MOVL C01095 V=800.0 PL=0
MOVL C01096 V=800.0 PL=0
MOVL C01097 V=800.0 PL=0
MOVL C01098 V=800.0 PL=0
MOVL C01099 V=800.0 PL=0
MOVL C01100 V=800.0 PL=0
MOVL C01101 V=800.0 PL=0
MOVL C01102 V=800.0 PL=0
MOVL C01103 V=800.0 PL=0
MOVL C01104 V=800.0 PL=0
MOVL C01105 V=800.0 PL=0
MOVL C01106 V=800.0 PL=0
MOVL C01107 V=800.0 PL=0
MOVL C01108 V=800.0 PL=0
MOVL C01109 V=800.0 PL=0
MOVL C01110 V=800.0 PL=0
MOVL C01111 V=800.0 PL=0
MOVL C01112 V=800.0 PL=0
MOVL C01113 V=800.0 PL=0
MOVL C01114 V=800.0 PL=0
MOVL C01115 V=800.0 PL=0
MOVL C01116 V=800.0 PL=0
MOVL C01117 V=800.0 PL=0
MOVL C01118 V=800.0 PL=0
MOVL C01119 V=800.0 PL=0
MOVL C01120 V=800.0 PL=0
MOVL C01121 V=800.0 PL=0
MOVL C01122 V=800.0 PL=0
MOVL C01123 V=800.0 PL=0
MOVL C01124 V=800.0 PL=0
MOVL C01125 V=800.0 PL=0
MOVL C01126 V=800.0 PL=0
MOVL C01127 V=800.0 PL=0
MOVL C01128 V=800.0 PL=0
MOVL C01129 V=800.0 PL=0
MOVL C01130 V=800.0 PL=0
MOVL C01131 V=800.0 PL=0
MOVL C01132 V=800.0 PL=0
MOVL C01133 V=800.0 PL=0
MOVL C01134 V=800.0 PL=0
MOVL C01135 V=800.0 PL=0
MOVL C01136 V=800.0 PL=0
MOVL C01137 V=800.0 PL=0
MOVL C01138 V=800.0 PL=0
MOVL C01139 V=800.0 PL=0
MOVL C01140 V=800.0 PL=0
MOVL C01141 V=800.0 PL=0
MOVL C01142 V=800.0 PL=0
MOVL C01143 V=800.0 PL=0
MOVL C01144 V=800.0 PL=0
MOVL C01145 V=800.0 PL=0
MOVL C01146 V=800.0 PL=0
MOVL C01147 V=800.0 PL=0
MOVL C01148 V=800.0 PL=0
MOVL C01149 V=800.0 PL=0
MOVL C01150 V=800.0 PL=0
MOVL C01151 V=800.0 PL=0
MOVL C01152 V=800.0 PL=0
MOVL C01153 V=800.0 PL=0
MOVL C01154 V=800.0 PL=0
MOVL C01155 V=800.0 PL=0
MOVL C01156 V=800.0 PL=0
MOVL C01157 V=800.0 PL=0
MOVL C01158 V=800.0 PL=0
MOVL C01159 V=800.0 PL=0
MOVL C01160 V=800.0 PL=0
MOVL C01161 V=800.0 PL=0
MOVL C01162 V=800.0 PL=0
MOVL C01163 V=800.0 PL=0
MOVL C01164 V=800.0 PL=0
MOVL C01165 V=800.0 PL=0
MOVL C01166 V=800.0 PL=0
MOVL C01167 V=800.0 PL=0
MOVL C01168 V=800.0 PL=0
MOVL C01169 V=800.0 PL=0
MOVL C01170 V=800.0 PL=0
MOVL C01171 V=800.0 PL=0
MOVL C01172 V=800.0 PL=0
MOVL C01173 V=800.0 PL=0
MOVL C01174 V=800.0 PL=0
MOVL C01175 V=800.0 PL=0
MOVL C01176 V=800.0 PL=0
MOVL C01177 V=800.0 PL=0
MOVL C01178 V=800.0 PL=0
MOVL C01179 V=800.0 PL=0
MOVL C01180 V=800.0 PL=0
MOVL C01181 V=800.0 PL=0
MOVL C01182 V=800.0 PL=0
MOVL C01183 V=800.0 PL=0
MOVL C01184 V=800.0 PL=0
MOVL C01185 V=800.0 PL=0
MOVL C01186 V=800.0 PL=0
MOVL C01187 V=800.0 PL=0
MOVL C01188 V=800.0 PL=0
MOVL C01189 V=800.0 PL=0
MOVL C01190 V=800.0 PL=0
MOVL C01191 V=800.0 PL=0
MOVL C01192 V=800.0 PL=0
MOVL C01193 V=800.0 PL=0
MOVL C01194 V=800.0 PL=0
MOVL C01195 V=800.0 PL=0
MOVL C01196 V=800.0 PL=0
MOVL C01197 V=800.0 PL=0
MOVL C01198 V=800.0 PL=0
MOVL C01199 V=800.0 PL=0
MOVL C01200 V=800.0 PL=0
MOVL C01201 V=800.0 PL=0
MOVL C01202 V=800.0 PL=0
MOVL C01203 V=800.0 PL=0
MOVL C01204 V=800.0 PL=0
MOVL C01205 V=800.0 PL=0
MOVL C01206 V=800.0 PL=0
MOVL C01207 V=800.0 PL=0
MOVL C01208 V=800.0 PL=0
MOVL C01209 V=800.0 PL=0
MOVL C01210 V=800.0 PL=0
MOVL C01211 V=800.0 PL=0
MOVL C01212 V=800.0 PL=0
MOVL C01213 V=800.0 PL=0
MOVL C01214 V=800.0 PL=0
MOVL C01215 V=800.0 PL=0
MOVL C01216 V=800.0 PL=0
MOVL C01217 V=800.0 PL=0
MOVL C01218 V=800.0 PL=0
MOVL C01219 V=800.0 PL=0
MOVL C01220 V=800.0 PL=0
MOVL C01221 V=800.0 PL=0
MOVL C01222 V=800.0 PL=0
MOVL C01223 V=800.0 PL=0
MOVL C01224 V=800.0 PL=0
MOVL C01225 V=800.0 PL=0
MOVL C01226 V=800.0 PL=0
MOVL C01227 V=800.0 PL=0
MOVL C01228 V=800.0 PL=0
MOVL C01229 V=800.0 PL=0
MOVL C01230 V=800.0 PL=0
MOVL C01231 V=800.0 PL=0
MOVL C01232 V=800.0 PL=0
MOVL C01233 V=800.0 PL=0
MOVL C01234 V=800.0 PL=0
MOVL C01235 V=800.0 PL=0
MOVL C01236 V=800.0 PL=0
MOVL C01237 V=800.0 PL=0
MOVL C01238 V=800.0 PL=0
MOVL C01239 V=800.0 PL=0
MOVL C01240 V=800.0 PL=0
MOVL C01241 V=800.0 PL=0
MOVL C01242 V=800.0 PL=0
MOVL C01243 V=800.0 PL=0
MOVL C01244 V=800.0 PL=0
MOVL C01245 V=800.0 PL=0
MOVL C01246 V=800.0 PL=0
MOVL C01247 V=800.0 PL=0
MOVL C01248 V=800.0 PL=0
MOVL C01249 V=800.0 PL=0
MOVL C01250 V=800.0 PL=0
MOVL C01251 V=800.0 PL=0
MOVL C01252 V=800.0 PL=0
MOVL C01253 V=800.0 PL=0
MOVL C01254 V=800.0 PL=0
MOVL C01255 V=800.0 PL=0
MOVL C01256 V=800.0 PL=0
MOVL C01257 V=800.0 PL=0
MOVL C01258 V=800.0 PL=0
MOVL C01259 V=800.0 PL=0
MOVL C01260 V=800.0 PL=0
MOVL C01261 V=800.0 PL=0
MOVL C01262 V=800.0 PL=0
MOVL C01263 V=800.0 PL=0
MOVL C01264 V=800.0 PL=0
MOVL C01265 V=800.0 PL=0
MOVL C01266 V=800.0 PL=0
MOVL C01267 V=800.0 PL=0
MOVL C01268 V=800.0 PL=0
MOVL C01269 V=800.0 PL=0
MOVL C01270 V=800.0 PL=0
MOVL C01271 V=800.0 PL=0
MOVL C01272 V=800.0 PL=0
MOVL C01273 V=800.0 PL=0
MOVL C01274 V=800.0 PL=0
MOVL C01275 V=800.0 PL=0
MOVL C01276 V=800.0 PL=0
MOVL C01277 V=800.0 PL=0
MOVL C01278 V=800.0 PL=0
MOVL C01279 V=800.0 PL=0
MOVL C01280 V=800.0 PL=0
MOVL C01281 V=800.0 PL=0
MOVL C01282 V=800.0 PL=0
MOVL C01283 V=800.0 PL=0
MOVL C01284 V=800.0 PL=0
MOVL C01285 V=800.0 PL=0
MOVL C01286 V=800.0 PL=0
MOVL C01287 V=800.0 PL=0
MOVL C01288 V=800.0 PL=0
MOVL C01289 V=800.0 PL=0
MOVL C01290 V=800.0 PL=0
MOVL C01291 V=800.0 PL=0
MOVL C01292 V=800.0 PL=0
MOVL C01293 V=800.0 PL=0
MOVL C01294 V=800.0 PL=0
MOVL C01295 V=800.0 PL=0
MOVL C01296 V=800.0 PL=0
MOVL C01297 V=800.0 PL=0
MOVL C01298 V=800.0 PL=0
MOVL C01299 V=800.0 PL=0
MOVL C01300 V=800.0 PL=0
MOVL C01301 V=800.0 PL=0
MOVL C01302 V=800.0 PL=0
MOVL C01303 V=800.0 PL=0
MOVL C01304 V=800.0 PL=0
MOVL C01305 V=800.0 PL=0
MOVL C01306 V=800.0 PL=0
MOVL C01307 V=800.0 PL=0
MOVL C01308 V=800.0 PL=0
MOVL C01309 V=800.0 PL=0
MOVL C01310 V=800.0 PL=0
MOVL C01311 V=800.0 PL=0
MOVL C01312 V=800.0 PL=0
MOVL C01313 V=800.0 PL=0
MOVL C01314 V=800.0 PL=0
MOVL C01315 V=800.0 PL=0
MOVL C01316 V=800.0 PL=0
MOVL C01317 V=800.0 PL=0
MOVL C01318 V=800.0 PL=0
MOVL C01319 V=800.0 PL=0
MOVL C01320 V=800.0 PL=0
MOVL C01321 V=800.0 PL=0
MOVL C01322 V=800.0 PL=0
MOVL C01323 V=800.0 PL=0
MOVL C01324 V=800.0 PL=0
MOVL C01325 V=800.0 PL=0
MOVL C01326 V=800.0 PL=0
MOVL C01327 V=800.0 PL=0
MOVL C01328 V=800.0 PL=0
MOVL C01329 V=800.0 PL=0
MOVL C01330 V=800.0 PL=0
MOVL C01331 V=800.0 PL=0
MOVL C01332 V=800.0 PL=0
MOVL C01333 V=800.0 PL=0
MOVL C01334 V=800.0 PL=0
MOVL C01335 V=800.0 PL=0
MOVL C01336 V=800.0 PL=0
MOVL C01337 V=800.0 PL=0
MOVL C01338 V=800.0 PL=0
MOVL C01339 V=800.0 PL=0
MOVL C01340 V=800.0 PL=0
MOVL C01341 V=800.0 PL=0
MOVL C01342 V=800.0 PL=0
MOVL C01343 V=800.0 PL=0
MOVL C01344 V=800.0 PL=0
MOVL C01345 V=800.0 PL=0
MOVL C01346 V=800.0 PL=0
MOVL C01347 V=800.0 PL=0
MOVL C01348 V=800.0 PL=0
MOVL C01349 V=800.0 PL=0
MOVL C01350 V=800.0 PL=0
MOVL C01351 V=800.0 PL=0
MOVL C01352 V=800.0 PL=0
MOVL C01353 V=800.0 PL=0
MOVL C01354 V=800.0 PL=0
MOVL C01355 V=800.0 PL=0
MOVL C01356 V=800.0 PL=0
MOVL C01357 V=800.0 PL=0
MOVL C01358 V=800.0 PL=0
MOVL C01359 V=800.0 PL=0
MOVL C01360 V=800.0 PL=0
MOVL C01361 V=800.0 PL=0
MOVL C01362 V=800.0 PL=0
MOVL C01363 V=800.0 PL=0
MOVL C01364 V=800.0 PL=0
MOVL C01365 V=800.0 PL=0
MOVL C01366 V=800.0 PL=0
MOVL C01367 V=800.0 PL=0
MOVL C01368 V=800.0 PL=0
MOVL C01369 V=800.0 PL=0
MOVL C01370 V=800.0 PL=0
MOVL C01371 V=800.0 PL=0
MOVL C01372 V=800.0 PL=0
MOVL C01373 V=800.0 PL=0
MOVL C01374 V=800.0 PL=0
MOVL C01375 V=800.0 PL=0
MOVL C01376 V=800.0 PL=0
MOVL C01377 V=800.0 PL=0
MOVL C01378 V=800.0 PL=0
MOVL C01379 V=800.0 PL=0
MOVL C01380 V=800.0 PL=0
MOVL C01381 V=800.0 PL=0
MOVL C01382 V=800.0 PL=0
MOVL C01383 V=800.0 PL=0
MOVL C01384 V=800.0 PL=0
MOVL C01385 V=800.0 PL=0
MOVL C01386 V=800.0 PL=0
MOVL C01387 V=800.0 PL=0
MOVL C01388 V=800.0 PL=0
MOVL C01389 V=800.0 PL=0
MOVL C01390 V=800.0 PL=0
MOVL C01391 V=800.0 PL=0
MOVL C01392 V=800.0 PL=0
MOVL C01393 V=800.0 PL=0
MOVL C01394 V=800.0 PL=0
MOVL C01395 V=800.0 PL=0
MOVL C01396 V=800.0 PL=0
MOVL C01397 V=800.0 PL=0
MOVL C01398 V=800.0 PL=0
MOVL C01399 V=800.0 PL=0
MOVL C01400 V=800.0 PL=0
MOVL C01401 V=800.0 PL=0
MOVL C01402 V=800.0 PL=0
MOVL C01403 V=800.0 PL=0
MOVL C01404 V=800.0 PL=0
MOVL C01405 V=800.0 PL=0
MOVL C01406 V=800.0 PL=0
MOVL C01407 V=800.0 PL=0
MOVL C01408 V=800.0 PL=0
MOVL C01409 V=800.0 PL=0
MOVL C01410 V=800.0 PL=0
MOVL C01411 V=800.0 PL=0
MOVL C01412 V=800.0 PL=0
MOVL C01413 V=800.0 PL=0
MOVL C01414 V=800.0 PL=0
MOVL C01415 V=800.0 PL=0
MOVL C01416 V=800.0 PL=0
MOVL C01417 V=800.0 PL=0
MOVL C01418 V=800.0 PL=0
MOVL C01419 V=800.0 PL=0
MOVL C01420 V=800.0 PL=0
MOVL C01421 V=800.0 PL=0
MOVL C01422 V=800.0 PL=0
MOVL C01423 V=800.0 PL=0
MOVL C01424 V=800.0 PL=0
MOVL C01425 V=800.0 PL=0
MOVL C01426 V=800.0 PL=0
MOVL C01427 V=800.0 PL=0
MOVL C01428 V=800.0 PL=0
MOVL C01429 V=800.0 PL=0
MOVL C01430 V=800.0 PL=0
MOVL C01431 V=800.0 PL=0
MOVL C01432 V=800.0 PL=0
MOVL C01433 V=800.0 PL=0
MOVL C01434 V=800.0 PL=0
MOVL C01435 V=800.0 PL=0
MOVL C01436 V=800.0 PL=0
MOVL C01437 V=800.0 PL=0
MOVL C01438 V=800.0 PL=0
MOVL C01439 V=800.0 PL=0
MOVL C01440 V=800.0 PL=0
MOVL C01441 V=800.0 PL=0
MOVL C01442 V=800.0 PL=0
MOVL C01443 V=800.0 PL=0
MOVL C01444 V=800.0 PL=0
MOVL C01445 V=800.0 PL=0
MOVL C01446 V=800.0 PL=0
MOVL C01447 V=800.0 PL=0
MOVL C01448 V=800.0 PL=0
MOVL C01449 V=800.0 PL=0
MOVL C01450 V=800.0 PL=0
MOVL C01451 V=800.0 PL=0
MOVL C01452 V=800.0 PL=0
MOVL C01453 V=800.0 PL=0
MOVL C01454 V=800.0 PL=0
MOVL C01455 V=800.0 PL=0
MOVL C01456 V=800.0 PL=0
MOVL C01457 V=800.0 PL=0
MOVL C01458 V=800.0 PL=0
MOVL C01459 V=800.0 PL=0
MOVL C01460 V=800.0 PL=0
MOVL C01461 V=800.0 PL=0
MOVL C01462 V=800.0 PL=0
MOVL C01463 V=800.0 PL=0
MOVL C01464 V=800.0 PL=0
MOVL C01465 V=800.0 PL=0
MOVL C01466 V=800.0 PL=0
MOVL C01467 V=800.0 PL=0
MOVL C01468 V=800.0 PL=0
MOVL C01469 V=800.0 PL=0
MOVL C01470 V=800.0 PL=0
MOVL C01471 V=800.0 PL=0
MOVL C01472 V=800.0 PL=0
MOVL C01473 V=800.0 PL=0
MOVL C01474 V=800.0 PL=0
MOVL C01475 V=800.0 PL=0
MOVL C01476 V=800.0 PL=0
MOVL C01477 V=800.0 PL=0
MOVL C01478 V=800.0 PL=0
MOVL C01479 V=800.0 PL=0
MOVL C01480 V=800.0 PL=0
MOVL C01481 V=800.0 PL=0
MOVL C01482 V=800.0 PL=0
MOVL C01483 V=800.0 PL=0
MOVL C01484 V=800.0 PL=0
MOVL C01485 V=800.0 PL=0
MOVL C01486 V=800.0 PL=0
MOVL C01487 V=800.0 PL=0
MOVL C01488 V=800.0 PL=0
MOVL C01489 V=800.0 PL=0
MOVL C01490 V=800.0 PL=0
MOVL C01491 V=800.0 PL=0
MOVL C01492 V=800.0 PL=0
MOVL C01493 V=800.0 PL=0
MOVL C01494 V=800.0 PL=0
MOVL C01495 V=800.0 PL=0
MOVL C01496 V=800.0 PL=0
MOVL C01497 V=800.0 PL=0
MOVL C01498 V=800.0 PL=0
MOVL C01499 V=800.0 PL=0
MOVL C01500 V=800.0 PL=0
MOVL C01501 V=800.0 PL=0
MOVL C01502 V=800.0 PL=0
MOVL C01503 V=800.0 PL=0
MOVL C01504 V=800.0 PL=0
MOVL C01505 V=800.0 PL=0
MOVL C01506 V=800.0 PL=0
MOVL C01507 V=800.0 PL=0
MOVL C01508 V=800.0 PL=0
MOVL C01509 V=800.0 PL=0
MOVL C01510 V=800.0 PL=0
MOVL C01511 V=800.0 PL=0
MOVL C01512 V=800.0 PL=0
MOVL C01513 V=800.0 PL=0
MOVL C01514 V=800.0 PL=0
MOVL C01515 V=800.0 PL=0
MOVL C01516 V=800.0 PL=0
MOVL C01517 V=800.0 PL=0
MOVL C01518 V=800.0 PL=0
MOVL C01519 V=800.0 PL=0
MOVL C01520 V=800.0 PL=0
MOVL C01521 V=800.0 PL=0
MOVL C01522 V=800.0 PL=0
MOVL C01523 V=800.0 PL=0
MOVL C01524 V=800.0 PL=0
MOVL C01525 V=800.0 PL=0
MOVL C01526 V=800.0 PL=0
MOVL C01527 V=800.0 PL=0
MOVL C01528 V=800.0 PL=0
MOVL C01529 V=800.0 PL=0
MOVL C01530 V=800.0 PL=0
MOVL C01531 V=800.0 PL=0
MOVL C01532 V=800.0 PL=0
MOVL C01533 V=800.0 PL=0
MOVL C01534 V=800.0 PL=0
MOVL C01535 V=800.0 PL=0
MOVL C01536 V=800.0 PL=0
MOVL C01537 V=800.0 PL=0
MOVL C01538 V=800.0 PL=0
MOVL C01539 V=800.0 PL=0
MOVL C01540 V=800.0 PL=0
MOVL C01541 V=800.0 PL=0
MOVL C01542 V=800.0 PL=0
MOVL C01543 V=800.0 PL=0
MOVL C01544 V=800.0 PL=0
MOVL C01545 V=800.0 PL=0
MOVL C01546 V=800.0 PL=0
MOVL C01547 V=800.0 PL=0
MOVL C01548 V=800.0 PL=0
MOVL C01549 V=800.0 PL=0
MOVL C01550 V=800.0 PL=0
MOVL C01551 V=800.0 PL=0
MOVL C01552 V=800.0 PL=0
MOVL C01553 V=800.0 PL=0
MOVL C01554 V=800.0 PL=0
MOVL C01555 V=800.0 PL=0
MOVL C01556 V=800.0 PL=0
MOVL C01557 V=800.0 PL=0
MOVL C01558 V=800.0 PL=0
MOVL C01559 V=800.0 PL=0
MOVL C01560 V=800.0 PL=0
MOVL C01561 V=800.0 PL=0
MOVL C01562 V=800.0 PL=0
MOVL C01563 V=800.0 PL=0
MOVL C01564 V=800.0 PL=0
MOVL C01565 V=800.0 PL=0
MOVL C01566 V=800.0 PL=0
MOVL C01567 V=800.0 PL=0
MOVL C01568 V=800.0 PL=0
MOVL C01569 V=800.0 PL=0
MOVL C01570 V=800.0 PL=0
MOVL C01571 V=800.0 PL=0
MOVL C01572 V=800.0 PL=0
MOVL C01573 V=800.0 PL=0
MOVL C01574 V=800.0 PL=0
MOVL C01575 V=800.0 PL=0
MOVL C01576 V=800.0 PL=0
MOVL C01577 V=800.0 PL=0
MOVL C01578 V=800.0 PL=0
MOVL C01579 V=800.0 PL=0
MOVL C01580 V=800.0 PL=0
MOVL C01581 V=800.0 PL=0
MOVL C01582 V=800.0 PL=0
MOVL C01583 V=800.0 PL=0
MOVL C01584 V=800.0 PL=0
MOVL C01585 V=800.0 PL=0
MOVL C01586 V=800.0 PL=0
MOVL C01587 V=800.0 PL=0
MOVL C01588 V=800.0 PL=0
MOVL C01589 V=800.0 PL=0
MOVL C01590 V=800.0 PL=0
MOVL C01591 V=800.0 PL=0
MOVL C01592 V=800.0 PL=0
MOVL C01593 V=800.0 PL=0
MOVL C01594 V=800.0 PL=0
MOVL C01595 V=800.0 PL=0
MOVL C01596 V=800.0 PL=0
MOVL C01597 V=800.0 PL=0
MOVL C01598 V=800.0 PL=0
MOVL C01599 V=800.0 PL=0
MOVL C01600 V=800.0 PL=0
MOVL C01601 V=800.0 PL=0
MOVL C01602 V=800.0 PL=0
MOVL C01603 V=800.0 PL=0
MOVL C01604 V=800.0 PL=0
MOVL C01605 V=800.0 PL=0
MOVL C01606 V=800.0 PL=0
MOVL C01607 V=800.0 PL=0
MOVL C01608 V=800.0 PL=0
MOVL C01609 V=800.0 PL=0
MOVL C01610 V=800.0 PL=0
MOVL C01611 V=800.0 PL=0
MOVL C01612 V=800.0 PL=0
MOVL C01613 V=800.0 PL=0
MOVL C01614 V=800.0 PL=0
MOVL C01615 V=800.0 PL=0
MOVL C01616 V=800.0 PL=0
MOVL C01617 V=800.0 PL=0
MOVL C01618 V=800.0 PL=0
MOVL C01619 V=800.0 PL=0
MOVL C01620 V=800.0 PL=0
MOVL C01621 V=800.0 PL=0
MOVL C01622 V=800.0 PL=0
MOVL C01623 V=800.0 PL=0
MOVL C01624 V=800.0 PL=0
MOVL C01625 V=800.0 PL=0
MOVL C01626 V=800.0 PL=0
MOVL C01627 V=800.0 PL=0
MOVL C01628 V=800.0 PL=0
MOVL C01629 V=800.0 PL=0
MOVL C01630 V=800.0 PL=0
MOVL C01631 V=800.0 PL=0
MOVL C01632 V=800.0 PL=0
MOVL C01633 V=800.0 PL=0
MOVL C01634 V=800.0 PL=0
MOVL C01635 V=800.0 PL=0
MOVL C01636 V=800.0 PL=0
MOVL C01637 V=800.0 PL=0
MOVL C01638 V=800.0 PL=0
MOVL C01639 V=800.0 PL=0
MOVL C01640 V=800.0 PL=0
MOVL C01641 V=800.0 PL=0
MOVL C01642 V=800.0 PL=0
MOVL C01643 V=800.0 PL=0
MOVL C01644 V=800.0 PL=0
MOVL C01645 V=800.0 PL=0
MOVL C01646 V=800.0 PL=0
MOVL C01647 V=800.0 PL=0
MOVL C01648 V=800.0 PL=0
MOVL C01649 V=800.0 PL=0
MOVL C01650 V=800.0 PL=0
MOVL C01651 V=800.0 PL=0
MOVL C01652 V=800.0 PL=0
MOVL C01653 V=800.0 PL=0
MOVL C01654 V=800.0 PL=0
MOVL C01655 V=800.0 PL=0
MOVL C01656 V=800.0 PL=0
MOVL C01657 V=800.0 PL=0
MOVL C01658 V=800.0 PL=0
MOVL C01659 V=800.0 PL=0
MOVL C01660 V=800.0 PL=0
MOVL C01661 V=800.0 PL=0
MOVL C01662 V=800.0 PL=0
MOVL C01663 V=800.0 PL=0
MOVL C01664 V=800.0 PL=0
MOVL C01665 V=800.0 PL=0
MOVL C01666 V=800.0 PL=0
MOVL C01667 V=800.0 PL=0
MOVL C01668 V=800.0 PL=0
MOVL C01669 V=800.0 PL=0
MOVL C01670 V=800.0 PL=0
MOVL C01671 V=800.0 PL=0
MOVL C01672 V=800.0 PL=0
MOVL C01673 V=800.0 PL=0
MOVL C01674 V=800.0 PL=0
MOVL C01675 V=800.0 PL=0
MOVL C01676 V=800.0 PL=0
MOVL C01677 V=800.0 PL=0
MOVL C01678 V=800.0 PL=0
MOVL C01679 V=800.0 PL=0
MOVL C01680 V=800.0 PL=0
MOVL C01681 V=800.0 PL=0
MOVL C01682 V=800.0 PL=0
MOVL C01683 V=800.0 PL=0
MOVL C01684 V=800.0 PL=0
MOVL C01685 V=800.0 PL=0
MOVL C01686 V=800.0 PL=0
MOVL C01687 V=800.0 PL=0
MOVL C01688 V=800.0 PL=0
MOVL C01689 V=800.0 PL=0
MOVL C01690 V=800.0 PL=0
MOVL C01691 V=800.0 PL=0
MOVL C01692 V=800.0 PL=0
MOVL C01693 V=800.0 PL=0
MOVL C01694 V=800.0 PL=0
MOVL C01695 V=800.0 PL=0
MOVL C01696 V=800.0 PL=0
MOVL C01697 V=800.0 PL=0
MOVL C01698 V=800.0 PL=0
MOVL C01699 V=800.0 PL=0
MOVL C01700 V=800.0 PL=0
MOVL C01701 V=800.0 PL=0
MOVL C01702 V=800.0 PL=0
MOVL C01703 V=800.0 PL=0
MOVL C01704 V=800.0 PL=0
MOVL C01705 V=800.0 PL=0
MOVL C01706 V=800.0 PL=0
MOVL C01707 V=800.0 PL=0
MOVL C01708 V=800.0 PL=0
MOVL C01709 V=800.0 PL=0
MOVL C01710 V=800.0 PL=0
MOVL C01711 V=800.0 PL=0
MOVL C01712 V=800.0 PL=0
MOVL C01713 V=800.0 PL=0
MOVL C01714 V=800.0 PL=0
MOVL C01715 V=800.0 PL=0
MOVL C01716 V=800.0 PL=0
MOVL C01717 V=800.0 PL=0
MOVL C01718 V=800.0 PL=0
MOVL C01719 V=800.0 PL=0
MOVL C01720 V=800.0 PL=0
MOVL C01721 V=800.0 PL=0
MOVL C01722 V=800.0 PL=0
MOVL C01723 V=800.0 PL=0
MOVL C01724 V=800.0 PL=0
MOVL C01725 V=800.0 PL=0
MOVL C01726 V=800.0 PL=0
MOVL C01727 V=800.0 PL=0
MOVL C01728 V=800.0 PL=0
MOVL C01729 V=800.0 PL=0
MOVL C01730 V=800.0 PL=0
MOVL C01731 V=800.0 PL=0
MOVL C01732 V=800.0 PL=0
MOVL C01733 V=800.0 PL=0
MOVL C01734 V=800.0 PL=0
MOVL C01735 V=800.0 PL=0
MOVL C01736 V=800.0 PL=0
MOVL C01737 V=800.0 PL=0
MOVL C01738 V=800.0 PL=0
MOVL C01739 V=800.0 PL=0
MOVL C01740 V=800.0 PL=0
MOVL C01741 V=800.0 PL=0
MOVL C01742 V=800.0 PL=0
MOVL C01743 V=800.0 PL=0
MOVL C01744 V=800.0 PL=0
MOVL C01745 V=800.0 PL=0
MOVL C01746 V=800.0 PL=0
MOVL C01747 V=800.0 PL=0
MOVL C01748 V=800.0 PL=0
MOVL C01749 V=800.0 PL=0
MOVL C01750 V=800.0 PL=0
MOVL C01751 V=800.0 PL=0
MOVL C01752 V=800.0 PL=0
MOVL C01753 V=800.0 PL=0
MOVL C01754 V=800.0 PL=0
MOVL C01755 V=800.0 PL=0
MOVL C01756 V=800.0 PL=0
MOVL C01757 V=800.0 PL=0
MOVL C01758 V=800.0 PL=0
MOVL C01759 V=800.0 PL=0
MOVL C01760 V=800.0 PL=0
MOVL C01761 V=800.0 PL=0
MOVL C01762 V=800.0 PL=0
MOVL C01763 V=800.0 PL=0
MOVL C01764 V=800.0 PL=0
MOVL C01765 V=800.0 PL=0
MOVL C01766 V=800.0 PL=0
MOVL C01767 V=800.0 PL=0
MOVL C01768 V=800.0 PL=0
MOVL C01769 V=800.0 PL=0
MOVL C01770 V=800.0 PL=0
MOVL C01771 V=800.0 PL=0
MOVL C01772 V=800.0 PL=0
MOVL C01773 V=800.0 PL=0
MOVL C01774 V=800.0 PL=0
MOVL C01775 V=800.0 PL=0
MOVL C01776 V=800.0 PL=0
MOVL C01777 V=800.0 PL=0
MOVL C01778 V=800.0 PL=0
MOVL C01779 V=800.0 PL=0
MOVL C01780 V=800.0 PL=0
MOVL C01781 V=800.0 PL=0
MOVL C01782 V=800.0 PL=0
MOVL C01783 V=800.0 PL=0
MOVL C01784 V=800.0 PL=0
MOVL C01785 V=800.0 PL=0
MOVL C01786 V=800.0 PL=0
MOVL C01787 V=800.0 PL=0
MOVL C01788 V=800.0 PL=0
MOVL C01789 V=800.0 PL=0
MOVL C01790 V=800.0 PL=0
MOVL C01791 V=800.0 PL=0
MOVL C01792 V=800.0 PL=0
MOVL C01793 V=800.0 PL=0
MOVL C01794 V=800.0 PL=0
MOVL C01795 V=800.0 PL=0
MOVL C01796 V=800.0 PL=0
MOVL C01797 V=800.0 PL=0
MOVL C01798 V=800.0 PL=0
MOVL C01799 V=800.0 PL=0
MOVL C01800 V=800.0 PL=0
MOVL C01801 V=800.0 PL=0
MOVL C01802 V=800.0 PL=0
MOVL C01803 V=800.0 PL=0
MOVL C01804 V=800.0 PL=0
MOVL C01805 V=800.0 PL=0
MOVL C01806 V=800.0 PL=0
MOVL C01807 V=800.0 PL=0
MOVL C01808 V=800.0 PL=0
MOVL C01809 V=800.0 PL=0
MOVL C01810 V=800.0 PL=0
MOVL C01811 V=800.0 PL=0
MOVL C01812 V=800.0 PL=0
MOVL C01813 V=800.0 PL=0
MOVL C01814 V=800.0 PL=0
MOVL C01815 V=800.0 PL=0
MOVL C01816 V=800.0 PL=0
MOVL C01817 V=800.0 PL=0
MOVL C01818 V=800.0 PL=0
MOVL C01819 V=800.0 PL=0
MOVL C01820 V=800.0 PL=0
MOVL C01821 V=800.0 PL=0
MOVL C01822 V=800.0 PL=0
MOVL C01823 V=800.0 PL=0
MOVL C01824 V=800.0 PL=0
MOVL C01825 V=800.0 PL=0
MOVL C01826 V=800.0 PL=0
MOVL C01827 V=800.0 PL=0
MOVL C01828 V=800.0 PL=0
MOVL C01829 V=800.0 PL=0
MOVL C01830 V=800.0 PL=0
MOVL C01831 V=800.0 PL=0
MOVL C01832 V=800.0 PL=0
MOVL C01833 V=800.0 PL=0
MOVL C01834 V=800.0 PL=0
MOVL C01835 V=800.0 PL=0
MOVL C01836 V=800.0 PL=0
MOVL C01837 V=800.0 PL=0
MOVL C01838 V=800.0 PL=0
MOVL C01839 V=800.0 PL=0
MOVL C01840 V=800.0 PL=0
MOVL C01841 V=800.0 PL=0
MOVL C01842 V=800.0 PL=0
MOVL C01843 V=800.0 PL=0
MOVL C01844 V=800.0 PL=0
MOVL C01845 V=800.0 PL=0
MOVL C01846 V=800.0 PL=0
MOVL C01847 V=800.0 PL=0
MOVL C01848 V=800.0 PL=0
MOVL C01849 V=800.0 PL=0
MOVL C01850 V=800.0 PL=0
MOVL C01851 V=800.0 PL=0
MOVL C01852 V=800.0 PL=0
MOVL C01853 V=800.0 PL=0
MOVL C01854 V=800.0 PL=0
MOVL C01855 V=800.0 PL=0
MOVL C01856 V=800.0 PL=0
MOVL C01857 V=800.0 PL=0
MOVL C01858 V=800.0 PL=0
MOVL C01859 V=800.0 PL=0
MOVL C01860 V=800.0 PL=0
MOVL C01861 V=800.0 PL=0
MOVL C01862 V=800.0 PL=0
MOVL C01863 V=800.0 PL=0
MOVL C01864 V=800.0 PL=0
MOVL C01865 V=800.0 PL=0
MOVL C01866 V=800.0 PL=0
MOVL C01867 V=800.0 PL=0
MOVL C01868 V=800.0 PL=0
MOVL C01869 V=800.0 PL=0
MOVL C01870 V=800.0 PL=0
MOVL C01871 V=800.0 PL=0
MOVL C01872 V=800.0 PL=0
MOVL C01873 V=800.0 PL=0
MOVL C01874 V=800.0 PL=0
MOVL C01875 V=800.0 PL=0
MOVL C01876 V=800.0 PL=0
MOVL C01877 V=800.0 PL=0
MOVL C01878 V=800.0 PL=0
MOVL C01879 V=800.0 PL=0
MOVL C01880 V=800.0 PL=0
MOVL C01881 V=800.0 PL=0
MOVL C01882 V=800.0 PL=0
MOVL C01883 V=800.0 PL=0
MOVL C01884 V=800.0 PL=0
MOVL C01885 V=800.0 PL=0
MOVL C01886 V=800.0 PL=0
MOVL C01887 V=800.0 PL=0
MOVL C01888 V=800.0 PL=0
MOVL C01889 V=800.0 PL=0
MOVL C01890 V=800.0 PL=0
MOVL C01891 V=800.0 PL=0
MOVL C01892 V=800.0 PL=0
MOVL C01893 V=800.0 PL=0
MOVL C01894 V=800.0 PL=0
MOVL C01895 V=800.0 PL=0
MOVL C01896 V=800.0 PL=0
MOVL C01897 V=800.0 PL=0
MOVL C01898 V=800.0 PL=0
MOVL C01899 V=800.0 PL=0
MOVL C01900 V=800.0 PL=0
MOVL C01901 V=800.0 PL=0
MOVL C01902 V=800.0 PL=0
MOVL C01903 V=800.0 PL=0
MOVL C01904 V=800.0 PL=0
MOVL C01905 V=800.0 PL=0
MOVL C01906 V=800.0 PL=0
MOVL C01907 V=800.0 PL=0
MOVL C01908 V=800.0 PL=0
MOVL C01909 V=800.0 PL=0
MOVL C01910 V=800.0 PL=0
MOVL C01911 V=800.0 PL=0
MOVL C01912 V=800.0 PL=0
MOVL C01913 V=800.0 PL=0
MOVL C01914 V=800.0 PL=0
MOVL C01915 V=800.0 PL=0
MOVL C01916 V=800.0 PL=0
MOVL C01917 V=800.0 PL=0
MOVL C01918 V=800.0 PL=0
MOVL C01919 V=800.0 PL=0
MOVL C01920 V=800.0 PL=0
MOVL C01921 V=800.0 PL=0
MOVL C01922 V=800.0 PL=0
MOVL C01923 V=800.0 PL=0
MOVL C01924 V=800.0 PL=0
MOVL C01925 V=800.0 PL=0
MOVL C01926 V=800.0 PL=0
MOVL C01927 V=800.0 PL=0
MOVL C01928 V=800.0 PL=0
MOVL C01929 V=800.0 PL=0
MOVL C01930 V=800.0 PL=0
MOVL C01931 V=800.0 PL=0
MOVL C01932 V=800.0 PL=0
MOVL C01933 V=800.0 PL=0
MOVL C01934 V=800.0 PL=0
MOVL C01935 V=800.0 PL=0
MOVL C01936 V=800.0 PL=0
MOVL C01937 V=800.0 PL=0
MOVL C01938 V=800.0 PL=0
MOVL C01939 V=800.0 PL=0
MOVL C01940 V=800.0 PL=0
MOVL C01941 V=800.0 PL=0
MOVL C01942 V=800.0 PL=0
MOVL C01943 V=800.0 PL=0
MOVL C01944 V=800.0 PL=0
MOVL C01945 V=800.0 PL=0
MOVL C01946 V=800.0 PL=0
MOVL C01947 V=800.0 PL=0
MOVL C01948 V=800.0 PL=0
MOVL C01949 V=800.0 PL=0
MOVL C01950 V=800.0 PL=0
MOVL C01951 V=800.0 PL=0
MOVL C01952 V=800.0 PL=0
MOVL C01953 V=800.0 PL=0
MOVL C01954 V=800.0 PL=0
MOVL C01955 V=800.0 PL=0
MOVL C01956 V=800.0 PL=0
MOVL C01957 V=800.0 PL=0
MOVL C01958 V=800.0 PL=0
MOVL C01959 V=800.0 PL=0
MOVL C01960 V=800.0 PL=0
MOVL C01961 V=800.0 PL=0
MOVL C01962 V=800.0 PL=0
MOVL C01963 V=800.0 PL=0
MOVL C01964 V=800.0 PL=0
MOVL C01965 V=800.0 PL=0
MOVL C01966 V=800.0 PL=0
MOVL C01967 V=800.0 PL=0
MOVL C01968 V=800.0 PL=0
MOVL C01969 V=800.0 PL=0
MOVL C01970 V=800.0 PL=0
MOVL C01971 V=800.0 PL=0
MOVL C01972 V=800.0 PL=0
MOVL C01973 V=800.0 PL=0
MOVL C01974 V=800.0 PL=0
MOVL C01975 V=800.0 PL=0
MOVL C01976 V=800.0 PL=0
MOVL C01977 V=800.0 PL=0
MOVL C01978 V=800.0 PL=0
MOVL C01979 V=800.0 PL=0
MOVL C01980 V=800.0 PL=0
MOVL C01981 V=800.0 PL=0
MOVL C01982 V=800.0 PL=0
MOVL C01983 V=800.0 PL=0
MOVL C01984 V=800.0 PL=0
MOVL C01985 V=800.0 PL=0
MOVL C01986 V=800.0 PL=0
MOVL C01987 V=800.0 PL=0
MOVL C01988 V=800.0 PL=0
MOVL C01989 V=800.0 PL=0
MOVL C01990 V=800.0 PL=0
MOVL C01991 V=800.0 PL=0
MOVL C01992 V=800.0 PL=0
MOVL C01993 V=800.0 PL=0
MOVL C01994 V=800.0 PL=0
MOVL C01995 V=800.0 PL=0
MOVL C01996 V=800.0 PL=0
MOVL C01997 V=800.0 PL=0
MOVL C01998 V=800.0 PL=0
MOVL C01999 V=800.0 PL=0
MOVL C02000 V=800.0 PL=0
MOVL C02001 V=800.0 PL=0
MOVL C02002 V=800.0 PL=0
MOVL C02003 V=800.0 PL=0
MOVL C02004 V=800.0 PL=0
MOVL C02005 V=800.0 PL=0
MOVL C02006 V=800.0 PL=0
MOVL C02007 V=800.0 PL=0
MOVL C02008 V=800.0 PL=0
MOVL C02009 V=800.0 PL=0
MOVL C02010 V=800.0 PL=0
MOVL C02011 V=800.0 PL=0
MOVL C02012 V=800.0 PL=0
MOVL C02013 V=800.0 PL=0
MOVL C02014 V=800.0 PL=0
MOVL C02015 V=800.0 PL=0
MOVL C02016 V=800.0 PL=0
MOVL C02017 V=800.0 PL=0
MOVL C02018 V=800.0 PL=0
MOVL C02019 V=800.0 PL=0
MOVL C02020 V=800.0 PL=0
MOVL C02021 V=800.0 PL=0
MOVL C02022 V=800.0 PL=0
MOVL C02023 V=800.0 PL=0
MOVL C02024 V=800.0 PL=0
MOVL C02025 V=800.0 PL=0
MOVL C02026 V=800.0 PL=0
MOVL C02027 V=800.0 PL=0
MOVL C02028 V=800.0 PL=0
MOVL C02029 V=800.0 PL=0
MOVL C02030 V=800.0 PL=0
MOVL C02031 V=800.0 PL=0
MOVL C02032 V=800.0 PL=0
MOVL C02033 V=800.0 PL=0
MOVL C02034 V=800.0 PL=0
MOVL C02035 V=800.0 PL=0
MOVL C02036 V=800.0 PL=0
MOVL C02037 V=800.0 PL=0
MOVL C02038 V=800.0 PL=0
MOVL C02039 V=800.0 PL=0
MOVL C02040 V=800.0 PL=0
MOVL C02041 V=800.0 PL=0
MOVL C02042 V=800.0 PL=0
MOVL C02043 V=800.0 PL=0
MOVL C02044 V=800.0 PL=0
MOVL C02045 V=800.0 PL=0
MOVL C02046 V=800.0 PL=0
MOVL C02047 V=800.0 PL=0
MOVL C02048 V=800.0 PL=0
MOVL C02049 V=800.0 PL=0
MOVL C02050 V=800.0 PL=0
MOVL C02051 V=800.0 PL=0
MOVL C02052 V=800.0 PL=0
MOVL C02053 V=800.0 PL=0
MOVL C02054 V=800.0 PL=0
MOVL C02055 V=800.0 PL=0
MOVL C02056 V=800.0 PL=0
MOVL C02057 V=800.0 PL=0
MOVL C02058 V=800.0 PL=0
MOVL C02059 V=800.0 PL=0
MOVL C02060 V=800.0 PL=0
MOVL C02061 V=800.0 PL=0
MOVL C02062 V=800.0 PL=0
MOVL C02063 V=800.0 PL=0
MOVL C02064 V=800.0 PL=0
MOVL C02065 V=800.0 PL=0
MOVL C02066 V=800.0 PL=0
MOVL C02067 V=800.0 PL=0
MOVL C02068 V=800.0 PL=0
MOVL C02069 V=800.0 PL=0
MOVL C02070 V=800.0 PL=0
MOVL C02071 V=800.0 PL=0
MOVL C02072 V=800.0 PL=0
MOVL C02073 V=800.0 PL=0
MOVL C02074 V=800.0 PL=0
MOVL C02075 V=800.0 PL=0
MOVL C02076 V=800.0 PL=0
MOVL C02077 V=800.0 PL=0
MOVL C02078 V=800.0 PL=0
MOVL C02079 V=800.0 PL=0
MOVL C02080 V=800.0 PL=0
MOVL C02081 V=800.0 PL=0
MOVL C02082 V=800.0 PL=0
MOVL C02083 V=800.0 PL=0
MOVL C02084 V=800.0 PL=0
MOVL C02085 V=800.0 PL=0
MOVL C02086 V=800.0 PL=0
MOVL C02087 V=800.0 PL=0
MOVL C02088 V=800.0 PL=0
MOVL C02089 V=800.0 PL=0
MOVL C02090 V=800.0 PL=0
MOVL C02091 V=800.0 PL=0
MOVL C02092 V=800.0 PL=0
MOVL C02093 V=800.0 PL=0
MOVL C02094 V=800.0 PL=0
MOVL C02095 V=800.0 PL=0
MOVL C02096 V=800.0 PL=0
MOVL C02097 V=800.0 PL=0
MOVL C02098 V=800.0 PL=0
MOVL C02099 V=800.0 PL=0
MOVL C02100 V=800.0 PL=0
MOVL C02101 V=800.0 PL=0
MOVL C02102 V=800.0 PL=0
MOVL C02103 V=800.0 PL=0
MOVL C02104 V=800.0 PL=0
MOVL C02105 V=800.0 PL=0
MOVL C02106 V=800.0 PL=0
MOVL C02107 V=800.0 PL=0
MOVL C02108 V=800.0 PL=0
MOVL C02109 V=800.0 PL=0
MOVL C02110 V=800.0 PL=0
MOVL C02111 V=800.0 PL=0
MOVL C02112 V=800.0 PL=0
MOVL C02113 V=800.0 PL=0
MOVL C02114 V=800.0 PL=0
MOVL C02115 V=800.0 PL=0
MOVL C02116 V=800.0 PL=0
MOVL C02117 V=800.0 PL=0
MOVL C02118 V=800.0 PL=0
MOVL C02119 V=800.0 PL=0
MOVL C02120 V=800.0 PL=0
MOVL C02121 V=800.0 PL=0
MOVL C02122 V=800.0 PL=0
MOVL C02123 V=800.0 PL=0
MOVL C02124 V=800.0 PL=0
MOVL C02125 V=800.0 PL=0
MOVL C02126 V=800.0 PL=0
MOVL C02127 V=800.0 PL=0
MOVL C02128 V=800.0 PL=0
MOVL C02129 V=800.0 PL=0
MOVL C02130 V=800.0 PL=0
MOVL C02131 V=800.0 PL=0
MOVL C02132 V=800.0 PL=0
MOVL C02133 V=800.0 PL=0
MOVL C02134 V=800.0 PL=0
MOVL C02135 V=800.0 PL=0
MOVL C02136 V=800.0 PL=0
MOVL C02137 V=800.0 PL=0
MOVL C02138 V=800.0 PL=0
MOVL C02139 V=800.0 PL=0
MOVL C02140 V=800.0 PL=0
MOVL C02141 V=800.0 PL=0
MOVL C02142 V=800.0 PL=0
MOVL C02143 V=800.0 PL=0
MOVL C02144 V=800.0 PL=0
MOVL C02145 V=800.0 PL=0
MOVL C02146 V=800.0 PL=0
MOVL C02147 V=800.0 PL=0
MOVL C02148 V=800.0 PL=0
MOVL C02149 V=800.0 PL=0
MOVL C02150 V=800.0 PL=0
MOVL C02151 V=800.0 PL=0
MOVL C02152 V=800.0 PL=0
MOVL C02153 V=800.0 PL=0
MOVL C02154 V=800.0 PL=0
MOVL C02155 V=800.0 PL=0
MOVL C02156 V=800.0 PL=0
MOVL C02157 V=800.0 PL=0
MOVL C02158 V=800.0 PL=0
MOVL C02159 V=800.0 PL=0
MOVL C02160 V=800.0 PL=0
MOVL C02161 V=800.0 PL=0
MOVL C02162 V=800.0 PL=0
MOVL C02163 V=800.0 PL=0
MOVL C02164 V=800.0 PL=0
MOVL C02165 V=800.0 PL=0
MOVL C02166 V=800.0 PL=0
MOVL C02167 V=800.0 PL=0
MOVL C02168 V=800.0 PL=0
MOVL C02169 V=800.0 PL=0
MOVL C02170 V=800.0 PL=0
MOVL C02171 V=800.0 PL=0
MOVL C02172 V=800.0 PL=0
MOVL C02173 V=800.0 PL=0
MOVL C02174 V=800.0 PL=0
